LIN {X -0.159,Y -541.286,Z 1239.781,A 0.000,B 0.000,C 90.000,E1 176.674} C_DIS
LIN {X -0.066,Y -543.209,Z 1239.777,A 0.000,B 0.000,C 90.000,E1 175.812} C_DIS
LIN {X 0.150,Y -546.405,Z 1239.769,A 0.000,B 0.000,C 90.000,E1 174.375} C_DIS
LIN {X -0.133,Y -549.421,Z 1239.761,A 0.000,B 0.000,C 90.000,E1 172.996} C_DIS
LIN {X -0.115,Y -552.819,Z 1239.752,A 0.000,B 0.000,C 90.000,E1 171.310} C_DIS
LIN {X -0.232,Y -555.615,Z 1239.744,A 0.000,B 0.000,C 90.000,E1 169.926} C_DIS
LIN {X -0.113,Y -558.230,Z 1239.736,A 0.000,B 0.000,C 90.000,E1 168.522} C_DIS
LIN {X 0.206,Y -561.440,Z 1239.727,A 0.000,B 0.000,C 90.000,E1 166.825} C_DIS
LIN {X -0.219,Y -565.186,Z 1239.716,A 0.000,B 0.000,C 90.000,E1 164.936} C_DIS
LIN {X 0.264,Y -570.650,Z 1239.703,A 0.000,B 0.000,C 90.000,E1 162.417} C_DIS
LIN {X -0.154,Y -576.138,Z 1239.692,A 0.000,B 0.000,C 90.000,E1 160.550} C_DIS
LIN {X 0.101,Y -582.010,Z 1239.683,A 0.000,B 0.000,C 90.000,E1 158.901} C_DIS
LIN {X -0.130,Y -586.378,Z 1239.677,A 0.000,B 0.000,C 90.000,E1 157.847} C_DIS
LIN {X 0.033,Y -593.495,Z 1239.668,A 0.000,B 0.000,C 90.000,E1 156.230} C_DIS
LIN {X -0.128,Y -599.475,Z 1239.661,A 0.000,B 0.000,C 90.000,E1 154.921} C_DIS
LIN {X 0.061,Y -605.395,Z 1239.653,A 0.000,B 0.000,C 90.000,E1 153.589} C_DIS
LIN {X 0.125,Y -609.959,Z 1239.648,A 0.000,B 0.000,C 90.000,E1 152.538} C_DIS
LIN {X -0.028,Y -614.349,Z 1239.642,A 0.000,B 0.000,C 90.000,E1 151.513} C_DIS
LIN {X 0.169,Y -618.559,Z 1239.636,A 0.000,B 0.000,C 90.000,E1 150.461} C_DIS
LIN {X -0.124,Y -624.838,Z 1239.627,A 0.000,B 0.000,C 90.000,E1 148.948} C_DIS
LIN {X 0.004,Y -628.846,Z 1239.622,A 0.000,B 0.000,C 90.000,E1 147.916} C_DIS
LIN {X -0.147,Y -632.777,Z 1239.616,A 0.000,B 0.000,C 90.000,E1 146.914} C_DIS
LIN {X -0.050,Y -637.321,Z 1239.609,A 0.000,B 0.000,C 90.000,E1 145.642} C_DIS
LIN {X 0.260,Y -640.796,Z 1239.604,A 0.000,B 0.000,C 90.000,E1 144.609} C_DIS
LIN {X 0.090,Y -643.931,Z 1239.598,A 0.000,B 0.000,C 90.000,E1 143.623} C_DIS
LIN {X -0.137,Y -647.459,Z 1239.591,A 0.000,B 0.000,C 90.000,E1 142.396} C_DIS
LIN {X 0.168,Y -650.146,Z 1239.586,A 0.000,B 0.000,C 90.000,E1 141.376} C_DIS
LIN {X -0.411,Y -652.643,Z 1239.580,A 0.000,B 0.000,C 90.000,E1 140.436} C_DIS
LIN {X -0.144,Y -656.271,Z 1239.572,A 0.000,B 0.000,C 90.000,E1 138.933} C_DIS
LIN {X -0.300,Y -659.807,Z 1239.564,A 0.000,B 0.000,C 90.000,E1 137.472} C_DIS
LIN {X 0.078,Y -662.638,Z 1239.557,A 0.000,B 0.000,C 90.000,E1 136.215} C_DIS
LIN {X 0.026,Y -668.777,Z 1239.543,A 0.000,B 0.000,C 90.000,E1 133.785} C_DIS
LIN {X 0.118,Y -672.513,Z 1239.535,A 0.000,B 0.000,C 90.000,E1 132.324} C_DIS
LIN {X -0.219,Y -676.296,Z 1239.527,A 0.000,B 0.000,C 90.000,E1 130.906} C_DIS
LIN {X 0.096,Y -680.057,Z 1239.519,A 0.000,B 0.000,C 90.000,E1 129.439} C_DIS
LIN {X -0.040,Y -683.726,Z 1239.511,A 0.000,B 0.000,C 90.000,E1 128.016} C_DIS
LIN {X 0.382,Y -686.776,Z 1239.505,A 0.000,B 0.000,C 90.000,E1 126.790} C_DIS
LIN {X -0.148,Y -689.067,Z 1239.499,A 0.000,B 0.000,C 90.000,E1 125.884} C_DIS
LIN {X -0.009,Y -692.235,Z 1239.491,A 0.000,B 0.000,C 90.000,E1 124.452} C_DIS
LIN {X -0.020,Y -695.390,Z 1239.484,A 0.000,B 0.000,C 90.000,E1 123.038} C_DIS
LIN {X -0.103,Y -696.843,Z 1239.480,A 0.000,B 0.000,C 90.000,E1 122.339} C_DIS
LIN {X 0.324,Y -699.079,Z 1239.473,A 0.000,B 0.000,C 90.000,E1 121.131} C_DIS
LIN {X -0.174,Y -701.315,Z 1239.467,A 0.000,B 0.000,C 90.000,E1 120.001} C_DIS
LIN {X -0.028,Y -703.175,Z 1239.460,A 0.000,B 0.000,C 90.000,E1 118.821} C_DIS
LIN {X 0.198,Y -704.139,Z 1239.456,A 0.000,B 0.000,C 90.000,E1 118.103} C_DIS
LIN {X 0.093,Y -705.071,Z 1239.451,A 0.000,B 0.000,C 90.000,E1 117.180} C_DIS
LIN {X 0.011,Y -705.580,Z 1239.447,A 0.000,B 0.000,C 90.000,E1 116.488} C_DIS
LIN {X -0.058,Y -705.835,Z 1239.443,A 0.000,B 0.000,C 90.000,E1 115.796} C_DIS
LIN {X 0.180,Y -705.686,Z 1239.439,A 0.000,B 0.000,C 90.000,E1 115.079} C_DIS
LIN {X -0.178,Y -705.329,Z 1239.437,A 0.000,B 0.000,C 90.000,E1 114.643} C_DIS
LIN {X 0.108,Y -704.589,Z 1239.434,A 0.000,B 0.000,C 90.000,E1 114.155} C_DIS
LIN {X -0.249,Y -704.115,Z 1239.433,A 0.000,B 0.000,C 90.000,E1 113.951} C_DIS
LIN {X 0.174,Y -701.663,Z 1239.430,A 0.000,B 0.000,C 90.000,E1 113.334} C_DIS
LIN {X 0.312,Y -700.871,Z 1239.429,A 0.000,B 0.000,C 90.000,E1 113.206} C_DIS
LIN {X 0.025,Y -696.095,Z 1239.427,A 0.000,B 0.000,C 90.000,E1 112.770} C_DIS
LIN {X 0.195,Y -694.683,Z 1239.426,A 0.000,B 0.000,C 90.000,E1 112.642} C_DIS
LIN {X 0.362,Y -692.329,Z 1239.425,A 0.000,B 0.000,C 90.000,E1 112.514} C_DIS
LIN {X 0.074,Y -686.037,Z 1239.424,A 0.000,B 0.000,C 90.000,E1 112.333} C_DIS
LIN {X -0.305,Y -683.624,Z 1239.424,A 0.000,B 0.000,C 90.000,E1 112.333} C_DIS
LIN {X -0.206,Y -677.436,Z 1239.424,A 0.000,B 0.000,C 90.000,E1 112.280} C_DIS
LIN {X -0.236,Y -621.471,Z 1239.424,A 0.000,B 0.000,C 90.000,E1 112.280} C_DIS
LIN {X 0.222,Y -618.148,Z 1239.422,A 0.000,B 0.000,C 90.000,E1 112.025} C_DIS
LIN {X -0.340,Y -616.389,Z 1239.421,A 0.000,B 0.000,C 90.000,E1 111.844} C_DIS
LIN {X -0.383,Y -616.380,Z 1239.421,A 0.000,B 0.000,C 90.000,E1 111.844} C_DIS
LIN {X -0.170,Y -616.270,Z 1239.420,A 0.000,B 0.000,C 90.000,E1 111.663} C_DIS
LIN {X -0.183,Y -616.646,Z 1239.420,A 0.000,B 0.000,C 90.000,E1 111.535} C_DIS
LIN {X 0.334,Y -618.749,Z 1239.417,A 0.000,B 0.000,C 90.000,E1 110.972} C_DIS
LIN {X -0.173,Y -622.755,Z 1239.412,A 0.000,B 0.000,C 90.000,E1 110.248} C_DIS
LIN {X 0.173,Y -625.249,Z 1239.410,A 0.000,B 0.000,C 90.000,E1 109.704} C_DIS
LIN {X -0.063,Y -628.625,Z 1239.405,A 0.000,B 0.000,C 90.000,E1 108.960} C_DIS
LIN {X -0.179,Y -640.008,Z 1239.391,A 0.000,B 0.000,C 90.000,E1 106.441} C_DIS
LIN {X 0.284,Y -642.172,Z 1239.389,A 0.000,B 0.000,C 90.000,E1 105.898} C_DIS
LIN {X -0.032,Y -644.177,Z 1239.386,A 0.000,B 0.000,C 90.000,E1 105.426} C_DIS
LIN {X -0.334,Y -646.007,Z 1239.383,A 0.000,B 0.000,C 90.000,E1 104.954} C_DIS
LIN {X 0.004,Y -647.639,Z 1239.380,A 0.000,B 0.000,C 90.000,E1 104.426} C_DIS
LIN {X -0.116,Y -648.936,Z 1239.377,A 0.000,B 0.000,C 90.000,E1 103.939} C_DIS
LIN {X 0.110,Y -650.550,Z 1239.373,A 0.000,B 0.000,C 90.000,E1 103.175} C_DIS
LIN {X -0.152,Y -651.298,Z 1239.371,A 0.000,B 0.000,C 90.000,E1 102.703} C_DIS
LIN {X 0.354,Y -651.536,Z 1239.369,A 0.000,B 0.000,C 90.000,E1 102.411} C_DIS
LIN {X -0.039,Y -651.751,Z 1239.366,A 0.000,B 0.000,C 90.000,E1 101.951} C_DIS
LIN {X -0.293,Y -651.502,Z 1239.364,A 0.000,B 0.000,C 90.000,E1 101.478} C_DIS
LIN {X 0.088,Y -650.980,Z 1239.361,A 0.000,B 0.000,C 90.000,E1 100.950} C_DIS
LIN {X -0.044,Y -650.643,Z 1239.359,A 0.000,B 0.000,C 90.000,E1 100.715} C_DIS
LIN {X 0.210,Y -649.651,Z 1239.357,A 0.000,B 0.000,C 90.000,E1 100.197} C_DIS
LIN {X -0.065,Y -648.276,Z 1239.354,A 0.000,B 0.000,C 90.000,E1 99.726} C_DIS
LIN {X 0.180,Y -646.565,Z 1239.351,A 0.000,B 0.000,C 90.000,E1 99.208} C_DIS
LIN {X -0.219,Y -644.492,Z 1239.349,A 0.000,B 0.000,C 90.000,E1 98.746} C_DIS
LIN {X 0.136,Y -642.730,Z 1239.346,A 0.000,B 0.000,C 90.000,E1 98.341} C_DIS
LIN {X -0.156,Y -640.829,Z 1239.344,A 0.000,B 0.000,C 90.000,E1 97.992} C_DIS
LIN {X -0.137,Y -636.009,Z 1239.340,A 0.000,B 0.000,C 90.000,E1 97.239} C_DIS
LIN {X 0.167,Y -633.458,Z 1239.338,A 0.000,B 0.000,C 90.000,E1 96.834} C_DIS
LIN {X 0.173,Y -628.255,Z 1239.335,A 0.000,B 0.000,C 90.000,E1 96.201} C_DIS
LIN {X -0.191,Y -625.016,Z 1239.333,A 0.000,B 0.000,C 90.000,E1 95.853} C_DIS
LIN {X -0.164,Y -617.303,Z 1239.328,A 0.000,B 0.000,C 90.000,E1 95.106} C_DIS
LIN {X -0.222,Y -610.306,Z 1239.325,A 0.000,B 0.000,C 90.000,E1 94.531} C_DIS
LIN {X -0.057,Y -604.326,Z 1239.323,A 0.000,B 0.000,C 90.000,E1 94.073} C_DIS
LIN {X 0.042,Y -596.685,Z 1239.320,A 0.000,B 0.000,C 90.000,E1 93.555} C_DIS
LIN {X 0.187,Y -586.971,Z 1239.317,A 0.000,B 0.000,C 90.000,E1 92.980} C_DIS
LIN {X 0.126,Y -583.659,Z 1239.316,A 0.000,B 0.000,C 90.000,E1 92.808} C_DIS
LIN {X -0.203,Y -576.652,Z 1239.314,A 0.000,B 0.000,C 90.000,E1 92.522} C_DIS
LIN {X -0.045,Y -571.225,Z 1239.313,A 0.000,B 0.000,C 90.000,E1 92.293} C_DIS
LIN {X -0.061,Y -567.337,Z 1239.312,A 0.000,B 0.000,C 90.000,E1 92.064} C_DIS
LIN {X 0.145,Y -566.878,Z 1239.311,A 0.000,B 0.000,C 90.000,E1 92.007} C_DIS
LIN {X -0.002,Y -566.188,Z 1239.311,A 0.000,B 0.000,C 90.000,E1 91.892} C_DIS
LIN {X -0.093,Y -566.019,Z 1239.306,A 0.000,B 0.000,C 90.000,E1 91.146} C_DIS
LIN {X 0.157,Y -567.324,Z 1239.296,A 0.000,B 0.000,C 90.000,E1 89.198} C_DIS
LIN {X -0.118,Y -568.765,Z 1239.285,A 0.000,B 0.000,C 90.000,E1 87.306} C_DIS
LIN {X 0.130,Y -571.142,Z 1239.270,A 0.000,B 0.000,C 90.000,E1 84.546} C_DIS
LIN {X -0.097,Y -572.726,Z 1239.261,A 0.000,B 0.000,C 90.000,E1 82.932} C_DIS
LIN {X -0.221,Y -574.365,Z 1239.252,A 0.000,B 0.000,C 90.000,E1 81.310} C_DIS
LIN {X -0.065,Y -575.384,Z 1239.246,A 0.000,B 0.000,C 90.000,E1 80.208} C_DIS
LIN {X -0.258,Y -576.370,Z 1239.238,A 0.000,B 0.000,C 90.000,E1 78.870} C_DIS
LIN {X 0.106,Y -577.627,Z 1239.228,A 0.000,B 0.000,C 90.000,E1 76.937} C_DIS
LIN {X -0.148,Y -578.654,Z 1239.219,A 0.000,B 0.000,C 90.000,E1 75.338} C_DIS
LIN {X -0.008,Y -579.712,Z 1239.208,A 0.000,B 0.000,C 90.000,E1 73.433} C_DIS
LIN {X -0.105,Y -580.316,Z 1239.202,A 0.000,B 0.000,C 90.000,E1 72.362} C_DIS
LIN {X -0.131,Y -581.509,Z 1239.192,A 0.000,B 0.000,C 90.000,E1 70.477} C_DIS
LIN {X 0.012,Y -582.379,Z 1239.182,A 0.000,B 0.000,C 90.000,E1 68.847} C_DIS
LIN {X 0.321,Y -584.062,Z 1239.171,A 0.000,B 0.000,C 90.000,E1 66.666} C_DIS
LIN {X -0.262,Y -585.676,Z 1239.160,A 0.000,B 0.000,C 90.000,E1 64.845} C_DIS
LIN {X 0.114,Y -587.635,Z 1239.148,A 0.000,B 0.000,C 90.000,E1 62.666} C_DIS
LIN {X 0.237,Y -589.240,Z 1239.139,A 0.000,B 0.000,C 90.000,E1 61.051} C_DIS
LIN {X 0.161,Y -590.895,Z 1239.130,A 0.000,B 0.000,C 90.000,E1 59.459} C_DIS
LIN {X 0.227,Y -592.252,Z 1239.123,A 0.000,B 0.000,C 90.000,E1 58.122} C_DIS
LIN {X -0.080,Y -593.318,Z 1239.117,A 0.000,B 0.000,C 90.000,E1 57.089} C_DIS
LIN {X 0.228,Y -594.723,Z 1239.108,A 0.000,B 0.000,C 90.000,E1 55.468} C_DIS
LIN {X -0.087,Y -596.078,Z 1239.099,A 0.000,B 0.000,C 90.000,E1 53.909} C_DIS
LIN {X 0.229,Y -597.028,Z 1239.092,A 0.000,B 0.000,C 90.000,E1 52.557} C_DIS
LIN {X -0.149,Y -597.936,Z 1239.086,A 0.000,B 0.000,C 90.000,E1 51.537} C_DIS
LIN {X 0.088,Y -598.439,Z 1239.082,A 0.000,B 0.000,C 90.000,E1 50.723} C_DIS
LIN {X 0.124,Y -599.217,Z 1239.073,A 0.000,B 0.000,C 90.000,E1 49.138} C_DIS
LIN {X 0.156,Y -599.656,Z 1239.067,A 0.000,B 0.000,C 90.000,E1 48.081} C_DIS
LIN {X -0.041,Y -599.960,Z 1239.063,A 0.000,B 0.000,C 90.000,E1 47.310} C_DIS
LIN {X -0.239,Y -600.183,Z 1239.058,A 0.000,B 0.000,C 90.000,E1 46.539} C_DIS
LIN {X 0.199,Y -600.293,Z 1239.050,A 0.000,B 0.000,C 90.000,E1 44.919} C_DIS
LIN {X 0.210,Y -600.158,Z 1239.044,A 0.000,B 0.000,C 90.000,E1 43.866} C_DIS
LIN {X 0.033,Y -599.798,Z 1239.036,A 0.000,B 0.000,C 90.000,E1 42.567} C_DIS
LIN {X 0.024,Y -599.344,Z 1239.031,A 0.000,B 0.000,C 90.000,E1 41.515} C_DIS
LIN {X 0.286,Y -598.606,Z 1239.023,A 0.000,B 0.000,C 90.000,E1 40.172} C_DIS
LIN {X 0.070,Y -598.239,Z 1239.019,A 0.000,B 0.000,C 90.000,E1 39.402} C_DIS
LIN {X -0.066,Y -597.699,Z 1239.015,A 0.000,B 0.000,C 90.000,E1 38.624} C_DIS
LIN {X -0.070,Y -596.650,Z 1239.009,A 0.000,B 0.000,C 90.000,E1 37.569} C_DIS
LIN {X 0.013,Y -595.473,Z 1239.003,A 0.000,B 0.000,C 90.000,E1 36.503} C_DIS
LIN {X -0.140,Y -594.382,Z 1238.998,A 0.000,B 0.000,C 90.000,E1 35.724} C_DIS
LIN {X -0.089,Y -592.672,Z 1238.993,A 0.000,B 0.000,C 90.000,E1 34.659} C_DIS
LIN {X -0.118,Y -591.215,Z 1238.988,A 0.000,B 0.000,C 90.000,E1 33.865} C_DIS
LIN {X 0.295,Y -590.086,Z 1238.985,A 0.000,B 0.000,C 90.000,E1 33.293} C_DIS
LIN {X -0.053,Y -587.340,Z 1238.979,A 0.000,B 0.000,C 90.000,E1 32.260} C_DIS
LIN {X -0.121,Y -585.016,Z 1238.975,A 0.000,B 0.000,C 90.000,E1 31.465} C_DIS
LIN {X -0.207,Y -582.273,Z 1238.970,A 0.000,B 0.000,C 90.000,E1 30.669} C_DIS
LIN {X -0.182,Y -580.238,Z 1238.967,A 0.000,B 0.000,C 90.000,E1 30.129} C_DIS
LIN {X 0.185,Y -576.738,Z 1238.963,A 0.000,B 0.000,C 90.000,E1 29.283} C_DIS
LIN {X 0.242,Y -574.841,Z 1238.961,A 0.000,B 0.000,C 90.000,E1 28.871} C_DIS
LIN {X 0.372,Y -569.197,Z 1238.955,A 0.000,B 0.000,C 90.000,E1 27.769} C_DIS
LIN {X -0.066,Y -565.217,Z 1238.951,A 0.000,B 0.000,C 90.000,E1 27.129} C_DIS
LIN {X 0.124,Y -560.088,Z 1238.946,A 0.000,B 0.000,C 90.000,E1 26.283} C_DIS
LIN {X 0.114,Y -555.294,Z 1238.942,A 0.000,B 0.000,C 90.000,E1 25.591} C_DIS
LIN {X 0.179,Y -551.321,Z 1238.939,A 0.000,B 0.000,C 90.000,E1 25.027} C_DIS
LIN {X 0.097,Y -545.830,Z 1238.935,A 0.000,B 0.000,C 90.000,E1 24.335} C_DIS
LIN {X 0.223,Y -542.367,Z 1238.933,A 0.000,B 0.000,C 90.000,E1 23.898} C_DIS
LIN {X 0.140,Y -532.373,Z 1238.927,A 0.000,B 0.000,C 90.000,E1 22.770} C_DIS
LIN {X 0.215,Y -528.501,Z 1238.924,A 0.000,B 0.000,C 90.000,E1 22.333} C_DIS
LIN {X -0.131,Y -519.371,Z 1238.919,A 0.000,B 0.000,C 90.000,E1 21.408} C_DIS
LIN {X 0.117,Y -508.642,Z 1238.913,A 0.000,B 0.000,C 90.000,E1 20.301} C_DIS
LIN {X -0.303,Y -498.892,Z 1238.908,A 0.000,B 0.000,C 90.000,E1 19.396} C_DIS
LIN {X 0.252,Y -489.022,Z 1238.903,A 0.000,B 0.000,C 90.000,E1 18.417} C_DIS
LIN {X 0.134,Y -480.227,Z 1238.898,A 0.000,B 0.000,C 90.000,E1 17.638} C_DIS
LIN {X -0.082,Y -465.601,Z 1238.891,A 0.000,B 0.000,C 90.000,E1 16.370} C_DIS
LIN {X -0.175,Y -443.465,Z 1238.880,A 0.000,B 0.000,C 90.000,E1 14.356} C_DIS
LIN {X -0.151,Y -424.558,Z 1238.869,A 0.000,B 0.000,C 90.000,E1 12.479} C_DIS
LIN {X -0.208,Y -403.283,Z 1238.856,A 0.000,B 0.000,C 90.000,E1 10.141} C_DIS
LIN {X 0.008,Y -399.230,Z 1238.854,A 0.000,B 0.000,C 90.000,E1 9.613} C_DIS
LIN {X -0.165,Y -396.098,Z 1238.851,A 0.000,B 0.000,C 90.000,E1 9.208} C_DIS
LIN {X 0.169,Y -395.193,Z 1238.850,A 0.000,B 0.000,C 90.000,E1 8.973} C_DIS
LIN {X 0.133,Y -394.246,Z 1238.849,A 0.000,B 0.000,C 90.000,E1 8.746} C_DIS
LIN {X 0.095,Y -394.236,Z 1238.849,A 0.000,B 0.000,C 90.000,E1 8.746} C_DIS
LIN {X -0.015,Y -394.164,Z 1238.848,A 0.000,B 0.000,C 90.000,E1 8.624} C_DIS
LIN {X -0.053,Y -394.166,Z 1238.848,A 0.000,B 0.000,C 90.000,E1 8.624} C_DIS
LIN {X 0.054,Y -396.357,Z 1238.845,A 0.000,B 0.000,C 90.000,E1 8.106} C_DIS
LIN {X 0.009,Y -397.853,Z 1238.844,A 0.000,B 0.000,C 90.000,E1 7.936} C_DIS
LIN {X -0.119,Y -400.874,Z 1238.842,A 0.000,B 0.000,C 90.000,E1 7.644} C_DIS
LIN {X 0.079,Y -406.596,Z 1238.840,A 0.000,B 0.000,C 90.000,E1 7.182} C_DIS
LIN {X -0.195,Y -414.525,Z 1238.837,A 0.000,B 0.000,C 90.000,E1 6.663} C_DIS
LIN {X 0.109,Y -422.610,Z 1238.834,A 0.000,B 0.000,C 90.000,E1 6.030} C_DIS
LIN {X -0.031,Y -430.604,Z 1238.830,A 0.000,B 0.000,C 90.000,E1 5.454} C_DIS
LIN {X -0.034,Y -443.124,Z 1238.825,A 0.000,B 0.000,C 90.000,E1 4.473} C_DIS
LIN {X -0.210,Y -457.129,Z 1238.819,A 0.000,B 0.000,C 90.000,E1 3.383} C_DIS
LIN {X -0.016,Y -463.216,Z 1238.816,A 0.000,B 0.000,C 90.000,E1 2.865} C_DIS
LIN {X 0.078,Y -469.211,Z 1238.813,A 0.000,B 0.000,C 90.000,E1 2.350} C_DIS
LIN {X 0.196,Y -473.636,Z 1238.811,A 0.000,B 0.000,C 90.000,E1 1.949} C_DIS
LIN {X 0.117,Y -479.358,Z 1238.808,A 0.000,B 0.000,C 90.000,E1 1.432} C_DIS
LIN {X -0.201,Y -484.890,Z 1238.805,A 0.000,B 0.000,C 90.000,E1 0.917} C_DIS
LIN {X -0.067,Y -491.548,Z 1238.801,A 0.000,B 0.000,C 90.000,E1 0.172} C_DIS
LIN {X 0.082,Y -497.345,Z 1238.797,A 0.000,B 0.000,C 90.000,E1 359.484} C_DIS
LIN {X 0.034,Y -503.232,Z 1238.793,A 0.000,B 0.000,C 90.000,E1 358.740} C_DIS
LIN {X 0.052,Y -508.653,Z 1238.789,A 0.000,B 0.000,C 90.000,E1 357.993} C_DIS
LIN {X 0.076,Y -513.670,Z 1238.785,A 0.000,B 0.000,C 90.000,E1 357.249} C_DIS
LIN {X 0.167,Y -518.402,Z 1238.781,A 0.000,B 0.000,C 90.000,E1 356.502} C_DIS
LIN {X 0.076,Y -521.935,Z 1238.777,A 0.000,B 0.000,C 90.000,E1 355.927} C_DIS
LIN {X 0.208,Y -525.937,Z 1238.773,A 0.000,B 0.000,C 90.000,E1 355.184} C_DIS
LIN {X -0.062,Y -529.601,Z 1238.769,A 0.000,B 0.000,C 90.000,E1 354.489} C_DIS
LIN {X -0.071,Y -532.321,Z 1238.766,A 0.000,B 0.000,C 90.000,E1 353.913} C_DIS
LIN {X -0.060,Y -534.872,Z 1238.763,A 0.000,B 0.000,C 90.000,E1 353.337} C_DIS
LIN {X -0.034,Y -537.243,Z 1238.760,A 0.000,B 0.000,C 90.000,E1 352.761} C_DIS
LIN {X 0.068,Y -540.450,Z 1238.755,A 0.000,B 0.000,C 90.000,E1 351.894} C_DIS
LIN {X 0.202,Y -543.387,Z 1238.750,A 0.000,B 0.000,C 90.000,E1 351.027} C_DIS
LIN {X -0.080,Y -546.130,Z 1238.746,A 0.000,B 0.000,C 90.000,E1 350.208} C_DIS
LIN {X -0.223,Y -550.100,Z 1238.738,A 0.000,B 0.000,C 90.000,E1 348.814} C_DIS
LIN {X -0.197,Y -553.570,Z 1238.730,A 0.000,B 0.000,C 90.000,E1 347.409} C_DIS
LIN {X -0.112,Y -556.059,Z 1238.724,A 0.000,B 0.000,C 90.000,E1 346.284} C_DIS
LIN {X -0.128,Y -558.246,Z 1238.718,A 0.000,B 0.000,C 90.000,E1 345.172} C_DIS
LIN {X 0.173,Y -560.272,Z 1238.711,A 0.000,B 0.000,C 90.000,E1 344.031} C_DIS
LIN {X -0.184,Y -562.020,Z 1238.705,A 0.000,B 0.000,C 90.000,E1 342.960} C_DIS
LIN {X 0.180,Y -563.501,Z 1238.699,A 0.000,B 0.000,C 90.000,E1 341.819} C_DIS
LIN {X 0.028,Y -564.723,Z 1238.693,A 0.000,B 0.000,C 90.000,E1 340.732} C_DIS
LIN {X 0.084,Y -565.529,Z 1238.687,A 0.000,B 0.000,C 90.000,E1 339.625} C_DIS
LIN {X -0.177,Y -565.847,Z 1238.682,A 0.000,B 0.000,C 90.000,E1 338.827} C_DIS
LIN {X -0.244,Y -565.913,Z 1238.679,A 0.000,B 0.000,C 90.000,E1 338.284} C_DIS
LIN {X 0.232,Y -565.700,Z 1238.675,A 0.000,B 0.000,C 90.000,E1 337.411} C_DIS
LIN {X -0.036,Y -565.160,Z 1238.670,A 0.000,B 0.000,C 90.000,E1 336.613} C_DIS
LIN {X 0.238,Y -563.873,Z 1238.664,A 0.000,B 0.000,C 90.000,E1 335.485} C_DIS
LIN {X -0.143,Y -563.050,Z 1238.661,A 0.000,B 0.000,C 90.000,E1 334.973} C_DIS
LIN {X -0.214,Y -561.509,Z 1238.656,A 0.000,B 0.000,C 90.000,E1 334.152} C_DIS
LIN {X 0.244,Y -558.987,Z 1238.650,A 0.000,B 0.000,C 90.000,E1 332.999} C_DIS
LIN {X 0.041,Y -558.330,Z 1238.649,A 0.000,B 0.000,C 90.000,E1 332.743} C_DIS
LIN {X -0.046,Y -554.735,Z 1238.642,A 0.000,B 0.000,C 90.000,E1 331.641} C_DIS
LIN {X 0.043,Y -551.366,Z 1238.638,A 0.000,B 0.000,C 90.000,E1 330.795} C_DIS
LIN {X -0.148,Y -548.734,Z 1238.635,A 0.000,B 0.000,C 90.000,E1 330.255} C_DIS
LIN {X 0.116,Y -545.883,Z 1238.632,A 0.000,B 0.000,C 90.000,E1 329.665} C_DIS
LIN {X -0.111,Y -542.741,Z 1238.628,A 0.000,B 0.000,C 90.000,E1 329.125} C_DIS
LIN {X 0.113,Y -537.269,Z 1238.624,A 0.000,B 0.000,C 90.000,E1 328.250} C_DIS
LIN {X 0.134,Y -532.378,Z 1238.620,A 0.000,B 0.000,C 90.000,E1 327.533} C_DIS
LIN {X -0.209,Y -526.129,Z 1238.615,A 0.000,B 0.000,C 90.000,E1 326.707} C_DIS
LIN {X -0.060,Y -518.520,Z 1238.609,A 0.000,B 0.000,C 90.000,E1 325.674} C_DIS
LIN {X 0.147,Y -514.711,Z 1238.606,A 0.000,B 0.000,C 90.000,E1 325.102} C_DIS
LIN {X -0.051,Y -511.652,Z 1238.603,A 0.000,B 0.000,C 90.000,E1 324.609} C_DIS
LIN {X -0.240,Y -508.815,Z 1238.600,A 0.000,B 0.000,C 90.000,E1 323.989} C_DIS
LIN {X 0.113,Y -506.962,Z 1238.596,A 0.000,B 0.000,C 90.000,E1 323.210} C_DIS
LIN {X -0.082,Y -506.057,Z 1238.592,A 0.000,B 0.000,C 90.000,E1 322.637} C_DIS
LIN {X 0.024,Y -505.470,Z 1238.589,A 0.000,B 0.000,C 90.000,E1 322.029} C_DIS
LIN {X -0.182,Y -505.207,Z 1238.586,A 0.000,B 0.000,C 90.000,E1 321.457} C_DIS
LIN {X -0.173,Y -506.208,Z 1238.571,A 0.000,B 0.000,C 90.000,E1 318.771} C_DIS
LIN {X 0.292,Y -506.801,Z 1238.563,A 0.000,B 0.000,C 90.000,E1 317.229} C_DIS
LIN {X -0.324,Y -507.316,Z 1238.554,A 0.000,B 0.000,C 90.000,E1 315.810} C_DIS
LIN {X -0.105,Y -507.935,Z 1238.543,A 0.000,B 0.000,C 90.000,E1 313.704} C_DIS
LIN {X 0.144,Y -508.691,Z 1238.531,A 0.000,B 0.000,C 90.000,E1 311.595} C_DIS
LIN {X 0.317,Y -509.214,Z 1238.523,A 0.000,B 0.000,C 90.000,E1 310.092} C_DIS
LIN {X 0.178,Y -509.639,Z 1238.515,A 0.000,B 0.000,C 90.000,E1 308.624} C_DIS
LIN {X 0.046,Y -510.089,Z 1238.506,A 0.000,B 0.000,C 90.000,E1 307.156} C_DIS
LIN {X 0.109,Y -510.410,Z 1238.500,A 0.000,B 0.000,C 90.000,E1 305.964} C_DIS
LIN {X 0.094,Y -510.717,Z 1238.492,A 0.000,B 0.000,C 90.000,E1 304.485} C_DIS
LIN {X 0.073,Y -511.002,Z 1238.484,A 0.000,B 0.000,C 90.000,E1 303.007} C_DIS
LIN {X -0.072,Y -511.155,Z 1238.475,A 0.000,B 0.000,C 90.000,E1 301.544} C_DIS
LIN {X 0.137,Y -511.238,Z 1238.465,A 0.000,B 0.000,C 90.000,E1 299.745} C_DIS
LIN {X -0.003,Y -511.239,Z 1238.457,A 0.000,B 0.000,C 90.000,E1 298.281} C_DIS
LIN {X 0.054,Y -511.208,Z 1238.449,A 0.000,B 0.000,C 90.000,E1 296.796} C_DIS
LIN {X 0.068,Y -511.329,Z 1238.434,A 0.000,B 0.000,C 90.000,E1 294.131} C_DIS
LIN {X 0.046,Y -511.394,Z 1238.428,A 0.000,B 0.000,C 90.000,E1 292.950} C_DIS
LIN {X 0.136,Y -510.947,Z 1238.419,A 0.000,B 0.000,C 90.000,E1 291.461} C_DIS
LIN {X -0.079,Y -510.463,Z 1238.413,A 0.000,B 0.000,C 90.000,E1 290.301} C_DIS
LIN {X -0.212,Y -509.464,Z 1238.400,A 0.000,B 0.000,C 90.000,E1 287.946} C_DIS
LIN {X -0.067,Y -509.112,Z 1238.395,A 0.000,B 0.000,C 90.000,E1 287.040} C_DIS
LIN {X 0.003,Y -508.188,Z 1238.383,A 0.000,B 0.000,C 90.000,E1 284.954} C_DIS
LIN {X 0.010,Y -507.302,Z 1238.375,A 0.000,B 0.000,C 90.000,E1 283.467} C_DIS
LIN {X -0.138,Y -506.650,Z 1238.370,A 0.000,B 0.000,C 90.000,E1 282.591} C_DIS
LIN {X 0.209,Y -506.076,Z 1238.365,A 0.000,B 0.000,C 90.000,E1 281.658} C_DIS
LIN {X 0.216,Y -504.023,Z 1238.350,A 0.000,B 0.000,C 90.000,E1 278.973} C_DIS
LIN {X -0.244,Y -503.117,Z 1238.342,A 0.000,B 0.000,C 90.000,E1 277.530} C_DIS
LIN {X 0.005,Y -501.816,Z 1238.328,A 0.000,B 0.000,C 90.000,E1 275.106} C_DIS
LIN {X -0.164,Y -500.807,Z 1238.318,A 0.000,B 0.000,C 90.000,E1 273.326} C_DIS
LIN {X -0.131,Y -500.000,Z 1238.312,A 0.000,B 0.000,C 90.000,E1 272.121} C_DIS
LIN {X -0.115,Y -499.040,Z 1238.305,A 0.000,B 0.000,C 90.000,E1 270.917} C_DIS
LIN {X -0.016,Y -497.609,Z 1238.293,A 0.000,B 0.000,C 90.000,E1 268.797} C_DIS
LIN {X 0.099,Y -497.010,Z 1238.288,A 0.000,B 0.000,C 90.000,E1 267.879} C_DIS
LIN {X -0.062,Y -496.196,Z 1238.280,A 0.000,B 0.000,C 90.000,E1 266.388} C_DIS
LIN {X 0.130,Y -495.162,Z 1238.270,A 0.000,B 0.000,C 90.000,E1 264.552} C_DIS
LIN {X -0.099,Y -493.875,Z 1238.260,A 0.000,B 0.000,C 90.000,E1 262.761} C_DIS
LIN {X -0.079,Y -492.806,Z 1238.253,A 0.000,B 0.000,C 90.000,E1 261.546} C_DIS
LIN {X -0.120,Y -490.157,Z 1238.238,A 0.000,B 0.000,C 90.000,E1 258.814} C_DIS
LIN {X 0.167,Y -488.574,Z 1238.226,A 0.000,B 0.000,C 90.000,E1 256.645} C_DIS
LIN {X 0.045,Y -487.272,Z 1238.214,A 0.000,B 0.000,C 90.000,E1 254.519} C_DIS
LIN {X 0.150,Y -485.968,Z 1238.202,A 0.000,B 0.000,C 90.000,E1 252.362} C_DIS
LIN {X -0.085,Y -484.912,Z 1238.190,A 0.000,B 0.000,C 90.000,E1 250.242} C_DIS
LIN {X -0.212,Y -484.287,Z 1238.183,A 0.000,B 0.000,C 90.000,E1 249.028} C_DIS
LIN {X -0.171,Y -483.475,Z 1238.175,A 0.000,B 0.000,C 90.000,E1 247.486} C_DIS
LIN {X 0.040,Y -482.481,Z 1238.166,A 0.000,B 0.000,C 90.000,E1 245.921} C_DIS
LIN {X -0.003,Y -481.068,Z 1238.156,A 0.000,B 0.000,C 90.000,E1 244.076} C_DIS
LIN {X -0.063,Y -479.930,Z 1238.147,A 0.000,B 0.000,C 90.000,E1 242.538} C_DIS
LIN {X 0.078,Y -478.591,Z 1238.139,A 0.000,B 0.000,C 90.000,E1 240.973} C_DIS
LIN {X -0.011,Y -477.472,Z 1238.132,A 0.000,B 0.000,C 90.000,E1 239.744} C_DIS
LIN {X 0.087,Y -475.588,Z 1238.122,A 0.000,B 0.000,C 90.000,E1 237.867} C_DIS
LIN {X 0.000,Y -473.771,Z 1238.111,A 0.000,B 0.000,C 90.000,E1 236.008} C_DIS
LIN {X 0.144,Y -472.113,Z 1238.101,A 0.000,B 0.000,C 90.000,E1 234.116} C_DIS
LIN {X -0.136,Y -470.493,Z 1238.090,A 0.000,B 0.000,C 90.000,E1 232.271} C_DIS
LIN {X -0.112,Y -468.614,Z 1238.078,A 0.000,B 0.000,C 90.000,E1 230.070} C_DIS
LIN {X 0.112,Y -466.861,Z 1238.066,A 0.000,B 0.000,C 90.000,E1 227.838} C_DIS
LIN {X -0.116,Y -465.418,Z 1238.055,A 0.000,B 0.000,C 90.000,E1 225.972} C_DIS
LIN {X -0.013,Y -463.787,Z 1238.034,A 0.000,B 0.000,C 90.000,E1 222.162} C_DIS
LIN {X -0.093,Y -465.130,Z 1237.997,A 0.000,B 0.000,C 90.000,E1 215.518} C_DIS
LIN {X 0.033,Y -468.440,Z 1237.973,A 0.000,B 0.000,C 90.000,E1 211.082} C_DIS
LIN {X -0.088,Y -472.228,Z 1237.954,A 0.000,B 0.000,C 90.000,E1 207.641} C_DIS
LIN {X -0.139,Y -474.591,Z 1237.943,A 0.000,B 0.000,C 90.000,E1 205.771} C_DIS
LIN {X -0.009,Y -479.495,Z 1237.924,A 0.000,B 0.000,C 90.000,E1 202.333} C_DIS
LIN {X -0.197,Y -485.542,Z 1237.905,A 0.000,B 0.000,C 90.000,E1 198.960} C_DIS
LIN {X -0.173,Y -492.217,Z 1237.888,A 0.000,B 0.000,C 90.000,E1 195.898} C_DIS
LIN {X -0.060,Y -496.543,Z 1237.878,A 0.000,B 0.000,C 90.000,E1 194.064} C_DIS
LIN {X 0.116,Y -500.278,Z 1237.870,A 0.000,B 0.000,C 90.000,E1 192.535} C_DIS
LIN {X 0.145,Y -505.606,Z 1237.858,A 0.000,B 0.000,C 90.000,E1 190.433} C_DIS
LIN {X -0.276,Y -511.238,Z 1237.847,A 0.000,B 0.000,C 90.000,E1 188.398} C_DIS
LIN {X -0.014,Y -515.254,Z 1237.838,A 0.000,B 0.000,C 90.000,E1 186.891} C_DIS
LIN {X 0.121,Y -520.743,Z 1237.827,A 0.000,B 0.000,C 90.000,E1 184.821} C_DIS
LIN {X -0.070,Y -524.642,Z 1237.819,A 0.000,B 0.000,C 90.000,E1 183.383} C_DIS
LIN {X -0.222,Y -528.511,Z 1237.811,A 0.000,B 0.000,C 90.000,E1 181.949} C_DIS
LIN {X 0.253,Y -530.814,Z 1237.806,A 0.000,B 0.000,C 90.000,E1 181.031} C_DIS
LIN {X 0.198,Y -534.608,Z 1237.798,A 0.000,B 0.000,C 90.000,E1 179.599} C_DIS
LIN {X 0.201,Y -537.567,Z 1237.792,A 0.000,B 0.000,C 90.000,E1 178.453} C_DIS
LIN {X 0.260,Y -540.380,Z 1237.785,A 0.000,B 0.000,C 90.000,E1 177.306} C_DIS
LIN {X -0.180,Y -543.140,Z 1237.779,A 0.000,B 0.000,C 90.000,E1 176.216} C_DIS
LIN {X 0.138,Y -547.659,Z 1237.768,A 0.000,B 0.000,C 90.000,E1 174.204} C_DIS
LIN {X -0.060,Y -550.679,Z 1237.760,A 0.000,B 0.000,C 90.000,E1 172.818} C_DIS
LIN {X -0.087,Y -554.231,Z 1237.751,A 0.000,B 0.000,C 90.000,E1 171.141} C_DIS
LIN {X -0.089,Y -557.072,Z 1237.743,A 0.000,B 0.000,C 90.000,E1 169.746} C_DIS
LIN {X 0.065,Y -559.775,Z 1237.735,A 0.000,B 0.000,C 90.000,E1 168.342} C_DIS
LIN {X -0.124,Y -563.074,Z 1237.726,A 0.000,B 0.000,C 90.000,E1 166.700} C_DIS
LIN {X -0.118,Y -566.420,Z 1237.717,A 0.000,B 0.000,C 90.000,E1 165.046} C_DIS
LIN {X 0.249,Y -572.000,Z 1237.703,A 0.000,B 0.000,C 90.000,E1 162.543} C_DIS
LIN {X -0.143,Y -577.479,Z 1237.693,A 0.000,B 0.000,C 90.000,E1 160.678} C_DIS
LIN {X 0.137,Y -583.215,Z 1237.684,A 0.000,B 0.000,C 90.000,E1 159.028} C_DIS
LIN {X 0.221,Y -589.838,Z 1237.675,A 0.000,B 0.000,C 90.000,E1 157.411} C_DIS
LIN {X 0.005,Y -595.701,Z 1237.667,A 0.000,B 0.000,C 90.000,E1 156.102} C_DIS
LIN {X -0.121,Y -601.578,Z 1237.660,A 0.000,B 0.000,C 90.000,E1 154.793} C_DIS
LIN {X 0.156,Y -606.242,Z 1237.654,A 0.000,B 0.000,C 90.000,E1 153.717} C_DIS
LIN {X -0.049,Y -610.732,Z 1237.648,A 0.000,B 0.000,C 90.000,E1 152.692} C_DIS
LIN {X 0.091,Y -615.025,Z 1237.643,A 0.000,B 0.000,C 90.000,E1 151.641} C_DIS
LIN {X 0.299,Y -619.154,Z 1237.637,A 0.000,B 0.000,C 90.000,E1 150.589} C_DIS
LIN {X 0.021,Y -625.228,Z 1237.628,A 0.000,B 0.000,C 90.000,E1 149.076} C_DIS
LIN {X 0.166,Y -630.145,Z 1237.621,A 0.000,B 0.000,C 90.000,E1 147.788} C_DIS
LIN {X 0.031,Y -633.889,Z 1237.616,A 0.000,B 0.000,C 90.000,E1 146.786} C_DIS
LIN {X 0.263,Y -636.554,Z 1237.611,A 0.000,B 0.000,C 90.000,E1 146.008} C_DIS
LIN {X 0.037,Y -640.008,Z 1237.606,A 0.000,B 0.000,C 90.000,E1 145.022} C_DIS
LIN {X -0.058,Y -641.677,Z 1237.603,A 0.000,B 0.000,C 90.000,E1 144.529} C_DIS
LIN {X -0.218,Y -644.675,Z 1237.597,A 0.000,B 0.000,C 90.000,E1 143.543} C_DIS
LIN {X 0.082,Y -648.118,Z 1237.590,A 0.000,B 0.000,C 90.000,E1 142.271} C_DIS
LIN {X -0.086,Y -651.340,Z 1237.584,A 0.000,B 0.000,C 90.000,E1 141.045} C_DIS
LIN {X -0.297,Y -654.312,Z 1237.577,A 0.000,B 0.000,C 90.000,E1 139.828} C_DIS
LIN {X -0.411,Y -656.689,Z 1237.571,A 0.000,B 0.000,C 90.000,E1 138.852} C_DIS
LIN {X -0.087,Y -659.620,Z 1237.564,A 0.000,B 0.000,C 90.000,E1 137.595} C_DIS
LIN {X -0.175,Y -663.007,Z 1237.556,A 0.000,B 0.000,C 90.000,E1 136.134} C_DIS
LIN {X -0.218,Y -669.111,Z 1237.543,A 0.000,B 0.000,C 90.000,E1 133.704} C_DIS
LIN {X -0.120,Y -672.855,Z 1237.535,A 0.000,B 0.000,C 90.000,E1 132.243} C_DIS
LIN {X 0.058,Y -676.610,Z 1237.527,A 0.000,B 0.000,C 90.000,E1 130.782} C_DIS
LIN {X -0.136,Y -680.348,Z 1237.519,A 0.000,B 0.000,C 90.000,E1 129.358} C_DIS
LIN {X -0.117,Y -684.611,Z 1237.509,A 0.000,B 0.000,C 90.000,E1 127.684} C_DIS
LIN {X -0.226,Y -687.628,Z 1237.503,A 0.000,B 0.000,C 90.000,E1 126.503} C_DIS
LIN {X -0.378,Y -689.328,Z 1237.499,A 0.000,B 0.000,C 90.000,E1 125.804} C_DIS
LIN {X 0.332,Y -692.498,Z 1237.491,A 0.000,B 0.000,C 90.000,E1 124.326} C_DIS
LIN {X 0.099,Y -695.153,Z 1237.484,A 0.000,B 0.000,C 90.000,E1 123.166} C_DIS
LIN {X 0.255,Y -697.081,Z 1237.479,A 0.000,B 0.000,C 90.000,E1 122.212} C_DIS
LIN {X 0.348,Y -699.778,Z 1237.471,A 0.000,B 0.000,C 90.000,E1 120.797} C_DIS
LIN {X 0.199,Y -701.523,Z 1237.466,A 0.000,B 0.000,C 90.000,E1 119.873} C_DIS
LIN {X -0.265,Y -703.436,Z 1237.460,A 0.000,B 0.000,C 90.000,E1 118.743} C_DIS
LIN {X 0.244,Y -704.592,Z 1237.454,A 0.000,B 0.000,C 90.000,E1 117.769} C_DIS
LIN {X -0.181,Y -705.446,Z 1237.449,A 0.000,B 0.000,C 90.000,E1 116.873} C_DIS
LIN {X 0.058,Y -705.814,Z 1237.445,A 0.000,B 0.000,C 90.000,E1 116.155} C_DIS
LIN {X -0.304,Y -705.935,Z 1237.443,A 0.000,B 0.000,C 90.000,E1 115.720} C_DIS
LIN {X -0.369,Y -705.725,Z 1237.439,A 0.000,B 0.000,C 90.000,E1 115.027} C_DIS
LIN {X 0.211,Y -705.341,Z 1237.436,A 0.000,B 0.000,C 90.000,E1 114.515} C_DIS
LIN {X -0.146,Y -704.549,Z 1237.434,A 0.000,B 0.000,C 90.000,E1 114.079} C_DIS
LIN {X 0.139,Y -703.840,Z 1237.432,A 0.000,B 0.000,C 90.000,E1 113.823} C_DIS
LIN {X -0.225,Y -701.803,Z 1237.430,A 0.000,B 0.000,C 90.000,E1 113.387} C_DIS
LIN {X -0.087,Y -701.068,Z 1237.429,A 0.000,B 0.000,C 90.000,E1 113.259} C_DIS
LIN {X -0.089,Y -698.721,Z 1237.428,A 0.000,B 0.000,C 90.000,E1 113.025} C_DIS
LIN {X -0.180,Y -695.031,Z 1237.426,A 0.000,B 0.000,C 90.000,E1 112.695} C_DIS
LIN {X -0.228,Y -693.057,Z 1237.425,A 0.000,B 0.000,C 90.000,E1 112.589} C_DIS
LIN {X 0.126,Y -686.215,Z 1237.424,A 0.000,B 0.000,C 90.000,E1 112.333} C_DIS
LIN {X -0.126,Y -685.182,Z 1237.424,A 0.000,B 0.000,C 90.000,E1 112.333} C_DIS
LIN {X -0.199,Y -677.161,Z 1237.424,A 0.000,B 0.000,C 90.000,E1 112.280} C_DIS
LIN {X -0.229,Y -620.472,Z 1237.424,A 0.000,B 0.000,C 90.000,E1 112.280} C_DIS
LIN {X 0.192,Y -617.806,Z 1237.423,A 0.000,B 0.000,C 90.000,E1 112.078} C_DIS
LIN {X -0.236,Y -616.859,Z 1237.422,A 0.000,B 0.000,C 90.000,E1 112.025} C_DIS
LIN {X -0.368,Y -615.087,Z 1237.421,A 0.000,B 0.000,C 90.000,E1 111.844} C_DIS
LIN {X 0.311,Y -614.938,Z 1237.421,A 0.000,B 0.000,C 90.000,E1 111.716} C_DIS
LIN {X -0.202,Y -614.914,Z 1237.420,A 0.000,B 0.000,C 90.000,E1 111.663} C_DIS
LIN {X -0.059,Y -615.601,Z 1237.419,A 0.000,B 0.000,C 90.000,E1 111.408} C_DIS
LIN {X -0.349,Y -617.782,Z 1237.416,A 0.000,B 0.000,C 90.000,E1 110.918} C_DIS
LIN {X -0.324,Y -620.311,Z 1237.413,A 0.000,B 0.000,C 90.000,E1 110.429} C_DIS
LIN {X -0.008,Y -623.432,Z 1237.410,A 0.000,B 0.000,C 90.000,E1 109.758} C_DIS
LIN {X 0.327,Y -626.747,Z 1237.406,A 0.000,B 0.000,C 90.000,E1 108.960} C_DIS
LIN {X 0.289,Y -631.542,Z 1237.399,A 0.000,B 0.000,C 90.000,E1 107.819} C_DIS
LIN {X -0.075,Y -635.615,Z 1237.394,A 0.000,B 0.000,C 90.000,E1 106.968} C_DIS
LIN {X -0.167,Y -640.139,Z 1237.389,A 0.000,B 0.000,C 90.000,E1 105.969} C_DIS
LIN {X -0.159,Y -641.185,Z 1237.387,A 0.000,B 0.000,C 90.000,E1 105.717} C_DIS
LIN {X -0.017,Y -643.975,Z 1237.383,A 0.000,B 0.000,C 90.000,E1 104.954} C_DIS
LIN {X -0.319,Y -645.507,Z 1237.380,A 0.000,B 0.000,C 90.000,E1 104.481} C_DIS
LIN {X 0.017,Y -646.945,Z 1237.378,A 0.000,B 0.000,C 90.000,E1 103.953} C_DIS
LIN {X 0.030,Y -647.523,Z 1237.376,A 0.000,B 0.000,C 90.000,E1 103.703} C_DIS
LIN {X 0.379,Y -648.467,Z 1237.373,A 0.000,B 0.000,C 90.000,E1 103.175} C_DIS
LIN {X -0.173,Y -649.559,Z 1237.369,A 0.000,B 0.000,C 90.000,E1 102.479} C_DIS
LIN {X 0.197,Y -649.786,Z 1237.367,A 0.000,B 0.000,C 90.000,E1 101.951} C_DIS
LIN {X -0.069,Y -649.528,Z 1237.364,A 0.000,B 0.000,C 90.000,E1 101.478} C_DIS
LIN {X 0.159,Y -648.612,Z 1237.360,A 0.000,B 0.000,C 90.000,E1 100.715} C_DIS
LIN {X -0.239,Y -647.597,Z 1237.357,A 0.000,B 0.000,C 90.000,E1 100.254} C_DIS
LIN {X 0.111,Y -646.208,Z 1237.354,A 0.000,B 0.000,C 90.000,E1 99.726} C_DIS
LIN {X -0.295,Y -644.508,Z 1237.351,A 0.000,B 0.000,C 90.000,E1 99.265} C_DIS
LIN {X -0.070,Y -642.452,Z 1237.349,A 0.000,B 0.000,C 90.000,E1 98.746} C_DIS
LIN {X -0.232,Y -641.312,Z 1237.347,A 0.000,B 0.000,C 90.000,E1 98.511} C_DIS
LIN {X -0.074,Y -637.841,Z 1237.344,A 0.000,B 0.000,C 90.000,E1 97.871} C_DIS
LIN {X -0.032,Y -633.863,Z 1237.340,A 0.000,B 0.000,C 90.000,E1 97.239} C_DIS
LIN {X 0.259,Y -631.201,Z 1237.338,A 0.000,B 0.000,C 90.000,E1 96.834} C_DIS
LIN {X 0.246,Y -625.976,Z 1237.335,A 0.000,B 0.000,C 90.000,E1 96.201} C_DIS
LIN {X -0.116,Y -622.416,Z 1237.333,A 0.000,B 0.000,C 90.000,E1 95.853} C_DIS
LIN {X 0.076,Y -617.407,Z 1237.330,A 0.000,B 0.000,C 90.000,E1 95.334} C_DIS
LIN {X -0.067,Y -610.497,Z 1237.326,A 0.000,B 0.000,C 90.000,E1 94.759} C_DIS
LIN {X 0.129,Y -603.034,Z 1237.323,A 0.000,B 0.000,C 90.000,E1 94.188} C_DIS
LIN {X -0.281,Y -595.216,Z 1237.321,A 0.000,B 0.000,C 90.000,E1 93.726} C_DIS
LIN {X 0.287,Y -584.228,Z 1237.317,A 0.000,B 0.000,C 90.000,E1 93.037} C_DIS
LIN {X 0.296,Y -580.414,Z 1237.316,A 0.000,B 0.000,C 90.000,E1 92.865} C_DIS
LIN {X -0.026,Y -571.859,Z 1237.314,A 0.000,B 0.000,C 90.000,E1 92.522} C_DIS
LIN {X 0.085,Y -566.784,Z 1237.313,A 0.000,B 0.000,C 90.000,E1 92.236} C_DIS
LIN {X 0.042,Y -566.759,Z 1237.313,A 0.000,B 0.000,C 90.000,E1 92.236} C_DIS
LIN {X -0.157,Y -566.349,Z 1237.312,A 0.000,B 0.000,C 90.000,E1 92.178} C_DIS
LIN {X 0.073,Y -565.918,Z 1237.311,A 0.000,B 0.000,C 90.000,E1 91.949} C_DIS
LIN {X 0.204,Y -565.846,Z 1237.309,A 0.000,B 0.000,C 90.000,E1 91.661} C_DIS
LIN {X -0.021,Y -566.103,Z 1237.305,A 0.000,B 0.000,C 90.000,E1 90.859} C_DIS
LIN {X 0.113,Y -567.281,Z 1237.296,A 0.000,B 0.000,C 90.000,E1 89.198} C_DIS
LIN {X -0.163,Y -568.704,Z 1237.285,A 0.000,B 0.000,C 90.000,E1 87.306} C_DIS
LIN {X -0.211,Y -570.516,Z 1237.273,A 0.000,B 0.000,C 90.000,E1 85.122} C_DIS
LIN {X 0.117,Y -572.128,Z 1237.264,A 0.000,B 0.000,C 90.000,E1 83.451} C_DIS
LIN {X 0.098,Y -574.013,Z 1237.253,A 0.000,B 0.000,C 90.000,E1 81.546} C_DIS
LIN {X -0.118,Y -575.259,Z 1237.246,A 0.000,B 0.000,C 90.000,E1 80.208} C_DIS
LIN {X 0.253,Y -576.231,Z 1237.238,A 0.000,B 0.000,C 90.000,E1 78.814} C_DIS
LIN {X 0.048,Y -577.492,Z 1237.228,A 0.000,B 0.000,C 90.000,E1 76.937} C_DIS
LIN {X -0.209,Y -578.504,Z 1237.219,A 0.000,B 0.000,C 90.000,E1 75.338} C_DIS
LIN {X 0.109,Y -579.394,Z 1237.209,A 0.000,B 0.000,C 90.000,E1 73.685} C_DIS
LIN {X 0.173,Y -580.032,Z 1237.203,A 0.000,B 0.000,C 90.000,E1 72.598} C_DIS
LIN {X 0.345,Y -581.356,Z 1237.192,A 0.000,B 0.000,C 90.000,E1 70.423} C_DIS
LIN {X -0.032,Y -583.453,Z 1237.174,A 0.000,B 0.000,C 90.000,E1 67.230} C_DIS
LIN {X -0.098,Y -585.074,Z 1237.163,A 0.000,B 0.000,C 90.000,E1 65.357} C_DIS
LIN {X -0.296,Y -586.436,Z 1237.154,A 0.000,B 0.000,C 90.000,E1 63.768} C_DIS
LIN {X 0.027,Y -587.511,Z 1237.148,A 0.000,B 0.000,C 90.000,E1 62.666} C_DIS
LIN {X 0.147,Y -589.118,Z 1237.139,A 0.000,B 0.000,C 90.000,E1 61.051} C_DIS
LIN {X 0.070,Y -590.781,Z 1237.130,A 0.000,B 0.000,C 90.000,E1 59.459} C_DIS
LIN {X 0.132,Y -592.121,Z 1237.123,A 0.000,B 0.000,C 90.000,E1 58.122} C_DIS
LIN {X -0.289,Y -593.388,Z 1237.116,A 0.000,B 0.000,C 90.000,E1 56.834} C_DIS
LIN {X 0.129,Y -594.574,Z 1237.108,A 0.000,B 0.000,C 90.000,E1 55.468} C_DIS
LIN {X 0.067,Y -595.681,Z 1237.101,A 0.000,B 0.000,C 90.000,E1 54.149} C_DIS
LIN {X -0.338,Y -596.505,Z 1237.095,A 0.000,B 0.000,C 90.000,E1 53.130} C_DIS
LIN {X -0.258,Y -597.767,Z 1237.086,A 0.000,B 0.000,C 90.000,E1 51.537} C_DIS
LIN {X -0.022,Y -598.279,Z 1237.082,A 0.000,B 0.000,C 90.000,E1 50.723} C_DIS
LIN {X 0.010,Y -599.028,Z 1237.073,A 0.000,B 0.000,C 90.000,E1 49.138} C_DIS
LIN {X 0.040,Y -599.500,Z 1237.067,A 0.000,B 0.000,C 90.000,E1 48.081} C_DIS
LIN {X -0.160,Y -599.789,Z 1237.063,A 0.000,B 0.000,C 90.000,E1 47.310} C_DIS
LIN {X 0.053,Y -600.011,Z 1237.058,A 0.000,B 0.000,C 90.000,E1 46.500} C_DIS
LIN {X 0.075,Y -600.119,Z 1237.050,A 0.000,B 0.000,C 90.000,E1 44.919} C_DIS
LIN {X 0.084,Y -599.972,Z 1237.044,A 0.000,B 0.000,C 90.000,E1 43.866} C_DIS
LIN {X 0.309,Y -599.605,Z 1237.036,A 0.000,B 0.000,C 90.000,E1 42.528} C_DIS
LIN {X -0.108,Y -599.125,Z 1237.031,A 0.000,B 0.000,C 90.000,E1 41.515} C_DIS
LIN {X 0.151,Y -598.396,Z 1237.023,A 0.000,B 0.000,C 90.000,E1 40.172} C_DIS
LIN {X -0.067,Y -598.023,Z 1237.019,A 0.000,B 0.000,C 90.000,E1 39.402} C_DIS
LIN {X -0.205,Y -597.473,Z 1237.015,A 0.000,B 0.000,C 90.000,E1 38.624} C_DIS
LIN {X 0.261,Y -596.412,Z 1237.009,A 0.000,B 0.000,C 90.000,E1 37.523} C_DIS
LIN {X -0.131,Y -595.219,Z 1237.003,A 0.000,B 0.000,C 90.000,E1 36.503} C_DIS
LIN {X 0.195,Y -594.114,Z 1236.998,A 0.000,B 0.000,C 90.000,E1 35.678} C_DIS
LIN {X 0.247,Y -592.403,Z 1236.992,A 0.000,B 0.000,C 90.000,E1 34.612} C_DIS
LIN {X 0.058,Y -590.916,Z 1236.988,A 0.000,B 0.000,C 90.000,E1 33.833} C_DIS
LIN {X 0.141,Y -589.780,Z 1236.985,A 0.000,B 0.000,C 90.000,E1 33.293} C_DIS
LIN {X 0.286,Y -587.031,Z 1236.979,A 0.000,B 0.000,C 90.000,E1 32.212} C_DIS
LIN {X -0.281,Y -584.670,Z 1236.975,A 0.000,B 0.000,C 90.000,E1 31.465} C_DIS
LIN {X -0.371,Y -581.895,Z 1236.970,A 0.000,B 0.000,C 90.000,E1 30.669} C_DIS
LIN {X 0.154,Y -579.850,Z 1236.967,A 0.000,B 0.000,C 90.000,E1 30.079} C_DIS
LIN {X 0.017,Y -576.306,Z 1236.963,A 0.000,B 0.000,C 90.000,E1 29.283} C_DIS
LIN {X 0.072,Y -574.417,Z 1236.960,A 0.000,B 0.000,C 90.000,E1 28.871} C_DIS
LIN {X 0.282,Y -569.470,Z 1236.955,A 0.000,B 0.000,C 90.000,E1 27.897} C_DIS
LIN {X -0.154,Y -565.567,Z 1236.951,A 0.000,B 0.000,C 90.000,E1 27.257} C_DIS
LIN {X 0.041,Y -560.451,Z 1236.947,A 0.000,B 0.000,C 90.000,E1 26.411} C_DIS
LIN {X 0.243,Y -557.650,Z 1236.944,A 0.000,B 0.000,C 90.000,E1 25.976} C_DIS
LIN {X 0.183,Y -551.870,Z 1236.940,A 0.000,B 0.000,C 90.000,E1 25.155} C_DIS
LIN {X 0.121,Y -546.442,Z 1236.936,A 0.000,B 0.000,C 90.000,E1 24.463} C_DIS
LIN {X -0.244,Y -543.040,Z 1236.934,A 0.000,B 0.000,C 90.000,E1 24.079} C_DIS
LIN {X 0.193,Y -533.109,Z 1236.927,A 0.000,B 0.000,C 90.000,E1 22.898} C_DIS
LIN {X 0.121,Y -527.912,Z 1236.924,A 0.000,B 0.000,C 90.000,E1 22.333} C_DIS
LIN {X 0.156,Y -518.656,Z 1236.919,A 0.000,B 0.000,C 90.000,E1 21.354} C_DIS
LIN {X -0.144,Y -509.172,Z 1236.913,A 0.000,B 0.000,C 90.000,E1 20.429} C_DIS
LIN {X -0.069,Y -497.882,Z 1236.907,A 0.000,B 0.000,C 90.000,E1 19.322} C_DIS
LIN {X 0.070,Y -487.659,Z 1236.902,A 0.000,B 0.000,C 90.000,E1 18.362} C_DIS
LIN {X 0.160,Y -480.328,Z 1236.898,A 0.000,B 0.000,C 90.000,E1 17.692} C_DIS
LIN {X -0.016,Y -465.932,Z 1236.891,A 0.000,B 0.000,C 90.000,E1 16.441} C_DIS
LIN {X 0.086,Y -444.036,Z 1236.880,A 0.000,B 0.000,C 90.000,E1 14.426} C_DIS
LIN {X -0.023,Y -425.326,Z 1236.870,A 0.000,B 0.000,C 90.000,E1 12.591} C_DIS
LIN {X -0.112,Y -403.997,Z 1236.857,A 0.000,B 0.000,C 90.000,E1 10.254} C_DIS
LIN {X 0.127,Y -399.903,Z 1236.854,A 0.000,B 0.000,C 90.000,E1 9.726} C_DIS
LIN {X 0.129,Y -395.849,Z 1236.851,A 0.000,B 0.000,C 90.000,E1 9.151} C_DIS
LIN {X -0.123,Y -394.216,Z 1236.849,A 0.000,B 0.000,C 90.000,E1 8.803} C_DIS
LIN {X -0.161,Y -394.207,Z 1236.849,A 0.000,B 0.000,C 90.000,E1 8.803} C_DIS
LIN {X 0.004,Y -394.134,Z 1236.848,A 0.000,B 0.000,C 90.000,E1 8.624} C_DIS
LIN {X -0.033,Y -394.135,Z 1236.848,A 0.000,B 0.000,C 90.000,E1 8.624} C_DIS
LIN {X 0.037,Y -396.432,Z 1236.845,A 0.000,B 0.000,C 90.000,E1 8.106} C_DIS
LIN {X -0.086,Y -398.558,Z 1236.844,A 0.000,B 0.000,C 90.000,E1 7.871} C_DIS
LIN {X 0.076,Y -401.188,Z 1236.842,A 0.000,B 0.000,C 90.000,E1 7.587} C_DIS
LIN {X -0.019,Y -408.232,Z 1236.839,A 0.000,B 0.000,C 90.000,E1 7.068} C_DIS
LIN {X 0.007,Y -414.743,Z 1236.837,A 0.000,B 0.000,C 90.000,E1 6.606} C_DIS
LIN {X 0.089,Y -425.581,Z 1236.832,A 0.000,B 0.000,C 90.000,E1 5.796} C_DIS
LIN {X -0.029,Y -431.899,Z 1236.830,A 0.000,B 0.000,C 90.000,E1 5.334} C_DIS
LIN {X -0.098,Y -444.478,Z 1236.824,A 0.000,B 0.000,C 90.000,E1 4.359} C_DIS
LIN {X -0.059,Y -456.788,Z 1236.819,A 0.000,B 0.000,C 90.000,E1 3.383} C_DIS
LIN {X 0.155,Y -462.865,Z 1236.816,A 0.000,B 0.000,C 90.000,E1 2.865} C_DIS
LIN {X -0.196,Y -468.933,Z 1236.813,A 0.000,B 0.000,C 90.000,E1 2.407} C_DIS
LIN {X -0.061,Y -473.350,Z 1236.811,A 0.000,B 0.000,C 90.000,E1 2.007} C_DIS
LIN {X -0.138,Y -479.096,Z 1236.808,A 0.000,B 0.000,C 90.000,E1 1.489} C_DIS
LIN {X 0.030,Y -484.689,Z 1236.805,A 0.000,B 0.000,C 90.000,E1 0.917} C_DIS
LIN {X -0.064,Y -491.166,Z 1236.801,A 0.000,B 0.000,C 90.000,E1 0.229} C_DIS
LIN {X 0.167,Y -497.428,Z 1236.797,A 0.000,B 0.000,C 90.000,E1 359.484} C_DIS
LIN {X 0.092,Y -503.378,Z 1236.793,A 0.000,B 0.000,C 90.000,E1 358.740} C_DIS
LIN {X 0.205,Y -508.789,Z 1236.789,A 0.000,B 0.000,C 90.000,E1 357.993} C_DIS
LIN {X 0.231,Y -513.881,Z 1236.785,A 0.000,B 0.000,C 90.000,E1 357.249} C_DIS
LIN {X -0.191,Y -518.620,Z 1236.781,A 0.000,B 0.000,C 90.000,E1 356.560} C_DIS
LIN {X 0.201,Y -522.162,Z 1236.778,A 0.000,B 0.000,C 90.000,E1 355.931} C_DIS
LIN {X 0.135,Y -525.472,Z 1236.774,A 0.000,B 0.000,C 90.000,E1 355.355} C_DIS
LIN {X -0.189,Y -529.220,Z 1236.770,A 0.000,B 0.000,C 90.000,E1 354.666} C_DIS
LIN {X 0.101,Y -532.631,Z 1236.766,A 0.000,B 0.000,C 90.000,E1 353.913} C_DIS
LIN {X 0.115,Y -535.186,Z 1236.763,A 0.000,B 0.000,C 90.000,E1 353.337} C_DIS
LIN {X 0.143,Y -537.556,Z 1236.760,A 0.000,B 0.000,C 90.000,E1 352.761} C_DIS
LIN {X 0.250,Y -540.771,Z 1236.755,A 0.000,B 0.000,C 90.000,E1 351.894} C_DIS
LIN {X -0.148,Y -543.743,Z 1236.750,A 0.000,B 0.000,C 90.000,E1 351.084} C_DIS
LIN {X 0.020,Y -545.585,Z 1236.747,A 0.000,B 0.000,C 90.000,E1 350.500} C_DIS
LIN {X -0.233,Y -548.870,Z 1236.741,A 0.000,B 0.000,C 90.000,E1 349.398} C_DIS
LIN {X 0.085,Y -551.165,Z 1236.736,A 0.000,B 0.000,C 90.000,E1 348.522} C_DIS
LIN {X 0.010,Y -553.906,Z 1236.730,A 0.000,B 0.000,C 90.000,E1 347.409} C_DIS
LIN {X -0.032,Y -556.396,Z 1236.724,A 0.000,B 0.000,C 90.000,E1 346.297} C_DIS
LIN {X 0.090,Y -558.615,Z 1236.718,A 0.000,B 0.000,C 90.000,E1 345.172} C_DIS
LIN {X -0.295,Y -560.669,Z 1236.712,A 0.000,B 0.000,C 90.000,E1 344.102} C_DIS
LIN {X 0.046,Y -562.424,Z 1236.705,A 0.000,B 0.000,C 90.000,E1 342.960} C_DIS
LIN {X -0.119,Y -563.935,Z 1236.699,A 0.000,B 0.000,C 90.000,E1 341.873} C_DIS
LIN {X 0.272,Y -565.217,Z 1236.693,A 0.000,B 0.000,C 90.000,E1 340.732} C_DIS
LIN {X 0.003,Y -565.879,Z 1236.689,A 0.000,B 0.000,C 90.000,E1 339.934} C_DIS
LIN {X -0.060,Y -566.234,Z 1236.686,A 0.000,B 0.000,C 90.000,E1 339.390} C_DIS
LIN {X 0.209,Y -566.471,Z 1236.681,A 0.000,B 0.000,C 90.000,E1 338.539} C_DIS
LIN {X -0.174,Y -566.513,Z 1236.678,A 0.000,B 0.000,C 90.000,E1 338.028} C_DIS
LIN {X 0.093,Y -566.251,Z 1236.673,A 0.000,B 0.000,C 90.000,E1 337.177} C_DIS
LIN {X 0.238,Y -565.914,Z 1236.670,A 0.000,B 0.000,C 90.000,E1 336.613} C_DIS
LIN {X 0.196,Y -565.033,Z 1236.666,A 0.000,B 0.000,C 90.000,E1 335.793} C_DIS
LIN {X 0.146,Y -563.912,Z 1236.661,A 0.000,B 0.000,C 90.000,E1 334.973} C_DIS
LIN {X -0.110,Y -561.838,Z 1236.655,A 0.000,B 0.000,C 90.000,E1 333.896} C_DIS
LIN {X -0.144,Y -559.288,Z 1236.649,A 0.000,B 0.000,C 90.000,E1 332.794} C_DIS
LIN {X -0.055,Y -557.570,Z 1236.646,A 0.000,B 0.000,C 90.000,E1 332.231} C_DIS
LIN {X 0.279,Y -555.795,Z 1236.643,A 0.000,B 0.000,C 90.000,E1 331.641} C_DIS
LIN {X -0.106,Y -552.460,Z 1236.638,A 0.000,B 0.000,C 90.000,E1 330.845} C_DIS
LIN {X 0.190,Y -549.877,Z 1236.635,A 0.000,B 0.000,C 90.000,E1 330.255} C_DIS
LIN {X -0.132,Y -546.316,Z 1236.631,A 0.000,B 0.000,C 90.000,E1 329.587} C_DIS
LIN {X 0.113,Y -543.131,Z 1236.628,A 0.000,B 0.000,C 90.000,E1 328.997} C_DIS
LIN {X -0.265,Y -538.565,Z 1236.624,A 0.000,B 0.000,C 90.000,E1 328.329} C_DIS
LIN {X 0.056,Y -533.669,Z 1236.620,A 0.000,B 0.000,C 90.000,E1 327.582} C_DIS
LIN {X 0.171,Y -527.426,Z 1236.615,A 0.000,B 0.000,C 90.000,E1 326.707} C_DIS
LIN {X -0.091,Y -517.650,Z 1236.608,A 0.000,B 0.000,C 90.000,E1 325.435} C_DIS
LIN {X 0.095,Y -514.607,Z 1236.605,A 0.000,B 0.000,C 90.000,E1 324.975} C_DIS
LIN {X -0.159,Y -511.962,Z 1236.603,A 0.000,B 0.000,C 90.000,E1 324.562} C_DIS
LIN {X -0.160,Y -509.626,Z 1236.600,A 0.000,B 0.000,C 90.000,E1 324.069} C_DIS
LIN {X 0.054,Y -508.682,Z 1236.599,A 0.000,B 0.000,C 90.000,E1 323.749} C_DIS
LIN {X 0.279,Y -507.167,Z 1236.595,A 0.000,B 0.000,C 90.000,E1 323.130} C_DIS
LIN {X -0.015,Y -505.952,Z 1236.590,A 0.000,B 0.000,C 90.000,E1 322.271} C_DIS
LIN {X -0.009,Y -505.452,Z 1236.585,A 0.000,B 0.000,C 90.000,E1 321.376} C_DIS
LIN {X 0.014,Y -506.557,Z 1236.571,A 0.000,B 0.000,C 90.000,E1 318.690} C_DIS
LIN {X -0.232,Y -507.181,Z 1236.562,A 0.000,B 0.000,C 90.000,E1 317.229} C_DIS
LIN {X -0.124,Y -507.696,Z 1236.554,A 0.000,B 0.000,C 90.000,E1 315.729} C_DIS
LIN {X -0.132,Y -508.290,Z 1236.544,A 0.000,B 0.000,C 90.000,E1 313.947} C_DIS
LIN {X 0.129,Y -509.025,Z 1236.533,A 0.000,B 0.000,C 90.000,E1 311.838} C_DIS
LIN {X 0.020,Y -509.489,Z 1236.526,A 0.000,B 0.000,C 90.000,E1 310.663} C_DIS
LIN {X -0.122,Y -510.001,Z 1236.518,A 0.000,B 0.000,C 90.000,E1 309.197} C_DIS
LIN {X -0.249,Y -510.416,Z 1236.510,A 0.000,B 0.000,C 90.000,E1 307.729} C_DIS
LIN {X 0.032,Y -510.851,Z 1236.501,A 0.000,B 0.000,C 90.000,E1 306.217} C_DIS
LIN {X 0.018,Y -511.206,Z 1236.493,A 0.000,B 0.000,C 90.000,E1 304.739} C_DIS
LIN {X 0.146,Y -511.550,Z 1236.485,A 0.000,B 0.000,C 90.000,E1 303.245} C_DIS
LIN {X -0.145,Y -511.691,Z 1236.477,A 0.000,B 0.000,C 90.000,E1 301.799} C_DIS
LIN {X 0.072,Y -511.825,Z 1236.467,A 0.000,B 0.000,C 90.000,E1 300.001} C_DIS
LIN {X -0.059,Y -511.873,Z 1236.458,A 0.000,B 0.000,C 90.000,E1 298.537} C_DIS
LIN {X 0.009,Y -511.857,Z 1236.450,A 0.000,B 0.000,C 90.000,E1 297.052} C_DIS
LIN {X -0.065,Y -511.922,Z 1236.437,A 0.000,B 0.000,C 90.000,E1 294.695} C_DIS
LIN {X 0.034,Y -512.066,Z 1236.429,A 0.000,B 0.000,C 90.000,E1 293.206} C_DIS
LIN {X -0.089,Y -511.886,Z 1236.424,A 0.000,B 0.000,C 90.000,E1 292.333} C_DIS
LIN {X 0.008,Y -511.420,Z 1236.416,A 0.000,B 0.000,C 90.000,E1 290.844} C_DIS
LIN {X -0.154,Y -510.577,Z 1236.406,A 0.000,B 0.000,C 90.000,E1 289.087} C_DIS
LIN {X 0.154,Y -509.954,Z 1236.396,A 0.000,B 0.000,C 90.000,E1 287.275} C_DIS
LIN {X 0.242,Y -508.975,Z 1236.385,A 0.000,B 0.000,C 90.000,E1 285.190} C_DIS
LIN {X 0.188,Y -508.259,Z 1236.378,A 0.000,B 0.000,C 90.000,E1 284.008} C_DIS
LIN {X 0.217,Y -507.947,Z 1236.375,A 0.000,B 0.000,C 90.000,E1 283.411} C_DIS
LIN {X -0.063,Y -506.737,Z 1236.365,A 0.000,B 0.000,C 90.000,E1 281.658} C_DIS
LIN {X 0.210,Y -504.182,Z 1236.345,A 0.000,B 0.000,C 90.000,E1 278.049} C_DIS
LIN {X -0.242,Y -503.250,Z 1236.337,A 0.000,B 0.000,C 90.000,E1 276.606} C_DIS
LIN {X 0.208,Y -502.342,Z 1236.327,A 0.000,B 0.000,C 90.000,E1 274.759} C_DIS
LIN {X 0.135,Y -501.491,Z 1236.318,A 0.000,B 0.000,C 90.000,E1 273.269} C_DIS
LIN {X -0.050,Y -500.205,Z 1236.308,A 0.000,B 0.000,C 90.000,E1 271.489} C_DIS
LIN {X 0.077,Y -498.652,Z 1236.297,A 0.000,B 0.000,C 90.000,E1 269.370} C_DIS
LIN {X -0.179,Y -498.253,Z 1236.293,A 0.000,B 0.000,C 90.000,E1 268.797} C_DIS
LIN {X 0.039,Y -497.200,Z 1236.283,A 0.000,B 0.000,C 90.000,E1 266.963} C_DIS
LIN {X 0.045,Y -496.525,Z 1236.276,A 0.000,B 0.000,C 90.000,E1 265.755} C_DIS
LIN {X 0.050,Y -495.829,Z 1236.270,A 0.000,B 0.000,C 90.000,E1 264.546} C_DIS
LIN {X -0.211,Y -494.536,Z 1236.260,A 0.000,B 0.000,C 90.000,E1 262.761} C_DIS
LIN {X 0.209,Y -493.171,Z 1236.251,A 0.000,B 0.000,C 90.000,E1 261.197} C_DIS
LIN {X -0.199,Y -490.806,Z 1236.238,A 0.000,B 0.000,C 90.000,E1 258.814} C_DIS
LIN {X 0.104,Y -489.219,Z 1236.226,A 0.000,B 0.000,C 90.000,E1 256.645} C_DIS
LIN {X -0.001,Y -487.912,Z 1236.214,A 0.000,B 0.000,C 90.000,E1 254.519} C_DIS
LIN {X 0.134,Y -486.427,Z 1236.200,A 0.000,B 0.000,C 90.000,E1 252.054} C_DIS
LIN {X -0.110,Y -485.724,Z 1236.192,A 0.000,B 0.000,C 90.000,E1 250.550} C_DIS
LIN {X -0.215,Y -484.951,Z 1236.183,A 0.000,B 0.000,C 90.000,E1 249.028} C_DIS
LIN {X -0.162,Y -484.124,Z 1236.175,A 0.000,B 0.000,C 90.000,E1 247.486} C_DIS
LIN {X 0.062,Y -483.106,Z 1236.166,A 0.000,B 0.000,C 90.000,E1 245.921} C_DIS
LIN {X 0.032,Y -481.691,Z 1236.156,A 0.000,B 0.000,C 90.000,E1 244.076} C_DIS
LIN {X -0.016,Y -480.540,Z 1236.147,A 0.000,B 0.000,C 90.000,E1 242.538} C_DIS
LIN {X 0.106,Y -478.905,Z 1236.137,A 0.000,B 0.000,C 90.000,E1 240.667} C_DIS
LIN {X 0.043,Y -477.364,Z 1236.129,A 0.000,B 0.000,C 90.000,E1 239.125} C_DIS
LIN {X 0.167,Y -476.092,Z 1236.122,A 0.000,B 0.000,C 90.000,E1 237.867} C_DIS
LIN {X 0.090,Y -474.273,Z 1236.111,A 0.000,B 0.000,C 90.000,E1 236.008} C_DIS
LIN {X 0.028,Y -472.202,Z 1236.099,A 0.000,B 0.000,C 90.000,E1 233.829} C_DIS
LIN {X -0.246,Y -471.343,Z 1236.094,A 0.000,B 0.000,C 90.000,E1 232.924} C_DIS
LIN {X 0.030,Y -469.652,Z 1236.083,A 0.000,B 0.000,C 90.000,E1 231.009} C_DIS
LIN {X -0.160,Y -468.310,Z 1236.075,A 0.000,B 0.000,C 90.000,E1 229.461} C_DIS
LIN {X -0.010,Y -466.822,Z 1236.064,A 0.000,B 0.000,C 90.000,E1 227.553} C_DIS
LIN {X 0.143,Y -465.218,Z 1236.052,A 0.000,B 0.000,C 90.000,E1 225.324} C_DIS
LIN {X -0.076,Y -463.771,Z 1236.031,A 0.000,B 0.000,C 90.000,E1 221.553} C_DIS
LIN {X 0.048,Y -465.188,Z 1235.997,A 0.000,B 0.000,C 90.000,E1 215.518} C_DIS
LIN {X -0.068,Y -468.742,Z 1235.971,A 0.000,B 0.000,C 90.000,E1 210.797} C_DIS
LIN {X 0.056,Y -472.191,Z 1235.954,A 0.000,B 0.000,C 90.000,E1 207.641} C_DIS
LIN {X -0.031,Y -474.924,Z 1235.942,A 0.000,B 0.000,C 90.000,E1 205.463} C_DIS
LIN {X 0.125,Y -479.982,Z 1235.922,A 0.000,B 0.000,C 90.000,E1 202.025} C_DIS
LIN {X -0.190,Y -486.782,Z 1235.902,A 0.000,B 0.000,C 90.000,E1 198.362} C_DIS
LIN {X -0.138,Y -492.925,Z 1235.887,A 0.000,B 0.000,C 90.000,E1 195.607} C_DIS
LIN {X -0.003,Y -497.324,Z 1235.877,A 0.000,B 0.000,C 90.000,E1 193.772} C_DIS
LIN {X 0.121,Y -501.890,Z 1235.867,A 0.000,B 0.000,C 90.000,E1 191.951} C_DIS
LIN {X 0.094,Y -508.999,Z 1235.852,A 0.000,B 0.000,C 90.000,E1 189.265} C_DIS
LIN {X -0.190,Y -513.123,Z 1235.843,A 0.000,B 0.000,C 90.000,E1 187.814} C_DIS
LIN {X 0.038,Y -517.099,Z 1235.835,A 0.000,B 0.000,C 90.000,E1 186.315} C_DIS
LIN {X -0.240,Y -521.896,Z 1235.825,A 0.000,B 0.000,C 90.000,E1 184.588} C_DIS
LIN {X 0.030,Y -527.416,Z 1235.814,A 0.000,B 0.000,C 90.000,E1 182.522} C_DIS
LIN {X -0.077,Y -531.315,Z 1235.806,A 0.000,B 0.000,C 90.000,E1 181.088} C_DIS
LIN {X -0.122,Y -534.403,Z 1235.800,A 0.000,B 0.000,C 90.000,E1 179.943} C_DIS
LIN {X -0.117,Y -538.151,Z 1235.792,A 0.000,B 0.000,C 90.000,E1 178.511} C_DIS
LIN {X -0.033,Y -541.709,Z 1235.784,A 0.000,B 0.000,C 90.000,E1 177.078} C_DIS
LIN {X 0.123,Y -544.438,Z 1235.777,A 0.000,B 0.000,C 90.000,E1 175.927} C_DIS
LIN {X -0.147,Y -548.403,Z 1235.768,A 0.000,B 0.000,C 90.000,E1 174.261} C_DIS
LIN {X 0.215,Y -551.479,Z 1235.760,A 0.000,B 0.000,C 90.000,E1 172.818} C_DIS
LIN {X 0.207,Y -555.128,Z 1235.751,A 0.000,B 0.000,C 90.000,E1 171.141} C_DIS
LIN {X -0.187,Y -558.608,Z 1235.742,A 0.000,B 0.000,C 90.000,E1 169.511} C_DIS
LIN {X -0.119,Y -561.425,Z 1235.734,A 0.000,B 0.000,C 90.000,E1 168.117} C_DIS
LIN {X -0.156,Y -564.856,Z 1235.725,A 0.000,B 0.000,C 90.000,E1 166.464} C_DIS
LIN {X 0.060,Y -568.961,Z 1235.714,A 0.000,B 0.000,C 90.000,E1 164.519} C_DIS
LIN {X 0.132,Y -576.564,Z 1235.697,A 0.000,B 0.000,C 90.000,E1 161.511} C_DIS
LIN {X -0.185,Y -580.894,Z 1235.690,A 0.000,B 0.000,C 90.000,E1 160.188} C_DIS
LIN {X -0.031,Y -585.800,Z 1235.682,A 0.000,B 0.000,C 90.000,E1 158.827} C_DIS
LIN {X -0.107,Y -595.889,Z 1235.669,A 0.000,B 0.000,C 90.000,E1 156.433} C_DIS
LIN {X 0.012,Y -601.598,Z 1235.662,A 0.000,B 0.000,C 90.000,E1 155.101} C_DIS
LIN {X 0.239,Y -607.325,Z 1235.654,A 0.000,B 0.000,C 90.000,E1 153.768} C_DIS
LIN {X 0.015,Y -612.755,Z 1235.647,A 0.000,B 0.000,C 90.000,E1 152.487} C_DIS
LIN {X 0.168,Y -617.906,Z 1235.640,A 0.000,B 0.000,C 90.000,E1 151.179} C_DIS
LIN {X -0.133,Y -623.833,Z 1235.631,A 0.000,B 0.000,C 90.000,E1 149.665} C_DIS
LIN {X 0.190,Y -627.814,Z 1235.626,A 0.000,B 0.000,C 90.000,E1 148.614} C_DIS
LIN {X 0.363,Y -631.580,Z 1235.620,A 0.000,B 0.000,C 90.000,E1 147.582} C_DIS
LIN {X 0.090,Y -636.117,Z 1235.613,A 0.000,B 0.000,C 90.000,E1 146.342} C_DIS
LIN {X -0.112,Y -640.325,Z 1235.606,A 0.000,B 0.000,C 90.000,E1 145.102} C_DIS
LIN {X -0.207,Y -641.979,Z 1235.603,A 0.000,B 0.000,C 90.000,E1 144.609} C_DIS
LIN {X 0.052,Y -645.612,Z 1235.596,A 0.000,B 0.000,C 90.000,E1 143.336} C_DIS
LIN {X -0.148,Y -648.932,Z 1235.589,A 0.000,B 0.000,C 90.000,E1 142.110} C_DIS
LIN {X -0.301,Y -652.028,Z 1235.583,A 0.000,B 0.000,C 90.000,E1 140.884} C_DIS
LIN {X 0.003,Y -654.962,Z 1235.576,A 0.000,B 0.000,C 90.000,E1 139.622} C_DIS
LIN {X -0.145,Y -657.872,Z 1235.569,A 0.000,B 0.000,C 90.000,E1 138.405} C_DIS
LIN {X 0.223,Y -660.177,Z 1235.563,A 0.000,B 0.000,C 90.000,E1 137.391} C_DIS
LIN {X -0.354,Y -664.131,Z 1235.554,A 0.000,B 0.000,C 90.000,E1 135.729} C_DIS
LIN {X -0.375,Y -669.028,Z 1235.543,A 0.000,B 0.000,C 90.000,E1 133.785} C_DIS
LIN {X -0.263,Y -673.387,Z 1235.534,A 0.000,B 0.000,C 90.000,E1 132.081} C_DIS
LIN {X -0.079,Y -677.115,Z 1235.526,A 0.000,B 0.000,C 90.000,E1 130.620} C_DIS
LIN {X 0.135,Y -680.196,Z 1235.519,A 0.000,B 0.000,C 90.000,E1 129.402} C_DIS
LIN {X 0.106,Y -683.859,Z 1235.511,A 0.000,B 0.000,C 90.000,E1 127.971} C_DIS
LIN {X -0.388,Y -687.489,Z 1235.503,A 0.000,B 0.000,C 90.000,E1 126.583} C_DIS
LIN {X -0.137,Y -689.202,Z 1235.499,A 0.000,B 0.000,C 90.000,E1 125.851} C_DIS
LIN {X 0.170,Y -692.398,Z 1235.491,A 0.000,B 0.000,C 90.000,E1 124.405} C_DIS
LIN {X -0.031,Y -695.551,Z 1235.483,A 0.000,B 0.000,C 90.000,E1 123.007} C_DIS
LIN {X 0.097,Y -697.001,Z 1235.479,A 0.000,B 0.000,C 90.000,E1 122.291} C_DIS
LIN {X 0.194,Y -699.724,Z 1235.472,A 0.000,B 0.000,C 90.000,E1 120.875} C_DIS
LIN {X 0.048,Y -701.472,Z 1235.466,A 0.000,B 0.000,C 90.000,E1 119.951} C_DIS
LIN {X -0.075,Y -703.053,Z 1235.461,A 0.000,B 0.000,C 90.000,E1 119.027} C_DIS
LIN {X -0.184,Y -704.389,Z 1235.456,A 0.000,B 0.000,C 90.000,E1 118.103} C_DIS
LIN {X 0.340,Y -705.275,Z 1235.451,A 0.000,B 0.000,C 90.000,E1 117.129} C_DIS
LIN {X -0.075,Y -705.881,Z 1235.446,A 0.000,B 0.000,C 90.000,E1 116.232} C_DIS
LIN {X -0.141,Y -706.002,Z 1235.442,A 0.000,B 0.000,C 90.000,E1 115.540} C_DIS
LIN {X -0.195,Y -705.895,Z 1235.439,A 0.000,B 0.000,C 90.000,E1 115.079} C_DIS
LIN {X 0.090,Y -705.541,Z 1235.437,A 0.000,B 0.000,C 90.000,E1 114.591} C_DIS
LIN {X 0.025,Y -704.779,Z 1235.434,A 0.000,B 0.000,C 90.000,E1 114.131} C_DIS
LIN {X 0.024,Y -704.265,Z 1235.433,A 0.000,B 0.000,C 90.000,E1 113.898} C_DIS
LIN {X -0.194,Y -701.560,Z 1235.430,A 0.000,B 0.000,C 90.000,E1 113.334} C_DIS
LIN {X -0.056,Y -700.687,Z 1235.429,A 0.000,B 0.000,C 90.000,E1 113.206} C_DIS
LIN {X -0.331,Y -695.836,Z 1235.426,A 0.000,B 0.000,C 90.000,E1 112.770} C_DIS
LIN {X -0.171,Y -694.255,Z 1235.426,A 0.000,B 0.000,C 90.000,E1 112.642} C_DIS
LIN {X -0.012,Y -691.473,Z 1235.425,A 0.000,B 0.000,C 90.000,E1 112.514} C_DIS
LIN {X 0.013,Y -685.813,Z 1235.424,A 0.000,B 0.000,C 90.000,E1 112.333} C_DIS
LIN {X 0.026,Y -679.669,Z 1235.424,A 0.000,B 0.000,C 90.000,E1 112.280} C_DIS
LIN {X -0.179,Y -676.996,Z 1235.424,A 0.000,B 0.000,C 90.000,E1 112.280} C_DIS
LIN {X -0.212,Y -619.525,Z 1235.424,A 0.000,B 0.000,C 90.000,E1 112.280} C_DIS
LIN {X 0.246,Y -616.043,Z 1235.422,A 0.000,B 0.000,C 90.000,E1 112.025} C_DIS
LIN {X -0.029,Y -614.093,Z 1235.421,A 0.000,B 0.000,C 90.000,E1 111.844} C_DIS
LIN {X -0.072,Y -614.076,Z 1235.421,A 0.000,B 0.000,C 90.000,E1 111.844} C_DIS
LIN {X 0.105,Y -613.609,Z 1235.420,A 0.000,B 0.000,C 90.000,E1 111.663} C_DIS
LIN {X 0.062,Y -613.609,Z 1235.420,A 0.000,B 0.000,C 90.000,E1 111.663} C_DIS
LIN {X -0.008,Y -614.361,Z 1235.419,A 0.000,B 0.000,C 90.000,E1 111.354} C_DIS
LIN {X -0.120,Y -615.589,Z 1235.417,A 0.000,B 0.000,C 90.000,E1 111.046} C_DIS
LIN {X -0.191,Y -618.131,Z 1235.414,A 0.000,B 0.000,C 90.000,E1 110.536} C_DIS
LIN {X -0.124,Y -621.819,Z 1235.410,A 0.000,B 0.000,C 90.000,E1 109.758} C_DIS
LIN {X 0.193,Y -625.016,Z 1235.406,A 0.000,B 0.000,C 90.000,E1 108.960} C_DIS
LIN {X 0.134,Y -629.147,Z 1235.400,A 0.000,B 0.000,C 90.000,E1 107.946} C_DIS
LIN {X 0.138,Y -634.880,Z 1235.393,A 0.000,B 0.000,C 90.000,E1 106.677} C_DIS
LIN {X -0.045,Y -636.031,Z 1235.391,A 0.000,B 0.000,C 90.000,E1 106.441} C_DIS
LIN {X -0.224,Y -638.135,Z 1235.389,A 0.000,B 0.000,C 90.000,E1 105.953} C_DIS
LIN {X 0.217,Y -639.312,Z 1235.387,A 0.000,B 0.000,C 90.000,E1 105.662} C_DIS
LIN {X -0.277,Y -641.952,Z 1235.383,A 0.000,B 0.000,C 90.000,E1 104.954} C_DIS
LIN {X 0.032,Y -643.523,Z 1235.380,A 0.000,B 0.000,C 90.000,E1 104.426} C_DIS
LIN {X 0.362,Y -645.478,Z 1235.376,A 0.000,B 0.000,C 90.000,E1 103.647} C_DIS
LIN {X 0.070,Y -646.442,Z 1235.373,A 0.000,B 0.000,C 90.000,E1 103.175} C_DIS
LIN {X -0.218,Y -647.132,Z 1235.370,A 0.000,B 0.000,C 90.000,E1 102.703} C_DIS
LIN {X -0.008,Y -647.556,Z 1235.368,A 0.000,B 0.000,C 90.000,E1 102.187} C_DIS
LIN {X -0.147,Y -647.639,Z 1235.366,A 0.000,B 0.000,C 90.000,E1 101.951} C_DIS
LIN {X 0.208,Y -647.502,Z 1235.364,A 0.000,B 0.000,C 90.000,E1 101.422} C_DIS
LIN {X -0.074,Y -646.869,Z 1235.361,A 0.000,B 0.000,C 90.000,E1 100.950} C_DIS
LIN {X 0.153,Y -645.906,Z 1235.358,A 0.000,B 0.000,C 90.000,E1 100.433} C_DIS
LIN {X 0.007,Y -645.345,Z 1235.357,A 0.000,B 0.000,C 90.000,E1 100.197} C_DIS
LIN {X 0.341,Y -643.951,Z 1235.354,A 0.000,B 0.000,C 90.000,E1 99.670} C_DIS
LIN {X -0.078,Y -642.156,Z 1235.351,A 0.000,B 0.000,C 90.000,E1 99.208} C_DIS
LIN {X -0.039,Y -638.705,Z 1235.347,A 0.000,B 0.000,C 90.000,E1 98.454} C_DIS
LIN {X 0.148,Y -635.999,Z 1235.344,A 0.000,B 0.000,C 90.000,E1 97.936} C_DIS
LIN {X -0.230,Y -632.961,Z 1235.341,A 0.000,B 0.000,C 90.000,E1 97.466} C_DIS
LIN {X -0.231,Y -628.301,Z 1235.338,A 0.000,B 0.000,C 90.000,E1 96.834} C_DIS
LIN {X 0.032,Y -625.347,Z 1235.336,A 0.000,B 0.000,C 90.000,E1 96.429} C_DIS
LIN {X -0.105,Y -617.989,Z 1235.332,A 0.000,B 0.000,C 90.000,E1 95.682} C_DIS
LIN {X 0.216,Y -612.539,Z 1235.329,A 0.000,B 0.000,C 90.000,E1 95.163} C_DIS
LIN {X 0.213,Y -608.250,Z 1235.327,A 0.000,B 0.000,C 90.000,E1 94.821} C_DIS
LIN {X -0.128,Y -602.283,Z 1235.324,A 0.000,B 0.000,C 90.000,E1 94.416} C_DIS
LIN {X 0.191,Y -597.645,Z 1235.323,A 0.000,B 0.000,C 90.000,E1 94.073} C_DIS
LIN {X -0.026,Y -589.814,Z 1235.320,A 0.000,B 0.000,C 90.000,E1 93.612} C_DIS
LIN {X -0.195,Y -583.207,Z 1235.318,A 0.000,B 0.000,C 90.000,E1 93.269} C_DIS
LIN {X -0.109,Y -579.688,Z 1235.317,A 0.000,B 0.000,C 90.000,E1 93.094} C_DIS
LIN {X 0.238,Y -571.011,Z 1235.315,A 0.000,B 0.000,C 90.000,E1 92.694} C_DIS
LIN {X -0.154,Y -567.214,Z 1235.314,A 0.000,B 0.000,C 90.000,E1 92.522} C_DIS
LIN {X -0.196,Y -567.142,Z 1235.314,A 0.000,B 0.000,C 90.000,E1 92.522} C_DIS
LIN {X 0.248,Y -566.162,Z 1235.313,A 0.000,B 0.000,C 90.000,E1 92.293} C_DIS
LIN {X 0.207,Y -566.147,Z 1235.313,A 0.000,B 0.000,C 90.000,E1 92.293} C_DIS
LIN {X -0.102,Y -566.061,Z 1235.312,A 0.000,B 0.000,C 90.000,E1 92.178} C_DIS
LIN {X 0.013,Y -565.660,Z 1235.311,A 0.000,B 0.000,C 90.000,E1 91.892} C_DIS
LIN {X 0.034,Y -566.280,Z 1235.303,A 0.000,B 0.000,C 90.000,E1 90.516} C_DIS
LIN {X 0.171,Y -567.477,Z 1235.294,A 0.000,B 0.000,C 90.000,E1 88.854} C_DIS
LIN {X 0.048,Y -569.143,Z 1235.282,A 0.000,B 0.000,C 90.000,E1 86.674} C_DIS
LIN {X 0.019,Y -571.040,Z 1235.269,A 0.000,B 0.000,C 90.000,E1 84.489} C_DIS
LIN {X -0.213,Y -572.638,Z 1235.260,A 0.000,B 0.000,C 90.000,E1 82.875} C_DIS
LIN {X 0.227,Y -574.228,Z 1235.251,A 0.000,B 0.000,C 90.000,E1 81.197} C_DIS
LIN {X 0.016,Y -575.388,Z 1235.244,A 0.000,B 0.000,C 90.000,E1 79.859} C_DIS
LIN {X -0.179,Y -576.326,Z 1235.236,A 0.000,B 0.000,C 90.000,E1 78.522} C_DIS
LIN {X -0.035,Y -577.402,Z 1235.227,A 0.000,B 0.000,C 90.000,E1 76.881} C_DIS
LIN {X 0.262,Y -578.391,Z 1235.218,A 0.000,B 0.000,C 90.000,E1 75.227} C_DIS
LIN {X 0.176,Y -579.279,Z 1235.209,A 0.000,B 0.000,C 90.000,E1 73.614} C_DIS
LIN {X -0.273,Y -580.058,Z 1235.202,A 0.000,B 0.000,C 90.000,E1 72.308} C_DIS
LIN {X 0.234,Y -581.237,Z 1235.191,A 0.000,B 0.000,C 90.000,E1 70.369} C_DIS
LIN {X -0.161,Y -583.356,Z 1235.173,A 0.000,B 0.000,C 90.000,E1 67.177} C_DIS
LIN {X 0.008,Y -584.987,Z 1235.163,A 0.000,B 0.000,C 90.000,E1 65.281} C_DIS
LIN {X -0.011,Y -587.197,Z 1235.149,A 0.000,B 0.000,C 90.000,E1 62.871} C_DIS
LIN {X -0.017,Y -589.054,Z 1235.139,A 0.000,B 0.000,C 90.000,E1 61.001} C_DIS
LIN {X 0.117,Y -590.148,Z 1235.133,A 0.000,B 0.000,C 90.000,E1 59.921} C_DIS
LIN {X -0.025,Y -591.282,Z 1235.127,A 0.000,B 0.000,C 90.000,E1 58.869} C_DIS
LIN {X 0.152,Y -592.291,Z 1235.121,A 0.000,B 0.000,C 90.000,E1 57.788} C_DIS
LIN {X -0.055,Y -593.792,Z 1235.112,A 0.000,B 0.000,C 90.000,E1 56.215} C_DIS
LIN {X -0.122,Y -594.936,Z 1235.105,A 0.000,B 0.000,C 90.000,E1 54.895} C_DIS
LIN {X 0.049,Y -596.179,Z 1235.096,A 0.000,B 0.000,C 90.000,E1 53.290} C_DIS
LIN {X -0.119,Y -597.633,Z 1235.086,A 0.000,B 0.000,C 90.000,E1 51.457} C_DIS
LIN {X 0.118,Y -598.144,Z 1235.081,A 0.000,B 0.000,C 90.000,E1 50.642} C_DIS
LIN {X -0.013,Y -599.007,Z 1235.071,A 0.000,B 0.000,C 90.000,E1 48.809} C_DIS
LIN {X 0.191,Y -599.596,Z 1235.064,A 0.000,B 0.000,C 90.000,E1 47.472} C_DIS
LIN {X -0.225,Y -599.837,Z 1235.058,A 0.000,B 0.000,C 90.000,E1 46.458} C_DIS
LIN {X -0.006,Y -599.935,Z 1235.051,A 0.000,B 0.000,C 90.000,E1 45.121} C_DIS
LIN {X 0.213,Y -599.765,Z 1235.043,A 0.000,B 0.000,C 90.000,E1 43.785} C_DIS
LIN {X 0.014,Y -599.561,Z 1235.039,A 0.000,B 0.000,C 90.000,E1 43.014} C_DIS
LIN {X 0.219,Y -599.243,Z 1235.035,A 0.000,B 0.000,C 90.000,E1 42.204} C_DIS
LIN {X 0.245,Y -598.720,Z 1235.029,A 0.000,B 0.000,C 90.000,E1 41.148} C_DIS
LIN {X 0.274,Y -597.934,Z 1235.020,A 0.000,B 0.000,C 90.000,E1 39.564} C_DIS
LIN {X -0.330,Y -597.429,Z 1235.016,A 0.000,B 0.000,C 90.000,E1 38.830} C_DIS
LIN {X 0.132,Y -596.389,Z 1235.010,A 0.000,B 0.000,C 90.000,E1 37.729} C_DIS
LIN {X -0.036,Y -594.884,Z 1235.002,A 0.000,B 0.000,C 90.000,E1 36.423} C_DIS
LIN {X 0.285,Y -593.763,Z 1234.998,A 0.000,B 0.000,C 90.000,E1 35.598} C_DIS
LIN {X -0.007,Y -592.011,Z 1234.992,A 0.000,B 0.000,C 90.000,E1 34.565} C_DIS
LIN {X -0.194,Y -590.465,Z 1234.988,A 0.000,B 0.000,C 90.000,E1 33.785} C_DIS
LIN {X 0.088,Y -588.681,Z 1234.983,A 0.000,B 0.000,C 90.000,E1 32.959} C_DIS
LIN {X 0.347,Y -586.573,Z 1234.979,A 0.000,B 0.000,C 90.000,E1 32.133} C_DIS
LIN {X 0.271,Y -584.106,Z 1234.974,A 0.000,B 0.000,C 90.000,E1 31.337} C_DIS
LIN {X 0.310,Y -582.312,Z 1234.971,A 0.000,B 0.000,C 90.000,E1 30.797} C_DIS
LIN {X 0.194,Y -579.187,Z 1234.967,A 0.000,B 0.000,C 90.000,E1 30.001} C_DIS
LIN {X 0.119,Y -576.195,Z 1234.963,A 0.000,B 0.000,C 90.000,E1 29.333} C_DIS
LIN {X -0.185,Y -573.656,Z 1234.960,A 0.000,B 0.000,C 90.000,E1 28.821} C_DIS
LIN {X 0.105,Y -569.374,Z 1234.956,A 0.000,B 0.000,C 90.000,E1 27.975} C_DIS
LIN {X -0.066,Y -565.535,Z 1234.952,A 0.000,B 0.000,C 90.000,E1 27.308} C_DIS
LIN {X -0.126,Y -560.411,Z 1234.947,A 0.000,B 0.000,C 90.000,E1 26.488} C_DIS
LIN {X -0.096,Y -554.896,Z 1234.943,A 0.000,B 0.000,C 90.000,E1 25.668} C_DIS
LIN {X 0.203,Y -550.900,Z 1234.939,A 0.000,B 0.000,C 90.000,E1 25.079} C_DIS
LIN {X 0.017,Y -544.229,Z 1234.935,A 0.000,B 0.000,C 90.000,E1 24.259} C_DIS
LIN {X 0.006,Y -538.350,Z 1234.931,A 0.000,B 0.000,C 90.000,E1 23.567} C_DIS
LIN {X 0.100,Y -530.947,Z 1234.926,A 0.000,B 0.000,C 90.000,E1 22.717} C_DIS
LIN {X -0.096,Y -521.864,Z 1234.921,A 0.000,B 0.000,C 90.000,E1 21.770} C_DIS
LIN {X -0.123,Y -517.834,Z 1234.919,A 0.000,B 0.000,C 90.000,E1 21.354} C_DIS
LIN {X 0.162,Y -508.486,Z 1234.913,A 0.000,B 0.000,C 90.000,E1 20.375} C_DIS
LIN {X 0.122,Y -497.555,Z 1234.907,A 0.000,B 0.000,C 90.000,E1 19.322} C_DIS
LIN {X -0.160,Y -488.791,Z 1234.903,A 0.000,B 0.000,C 90.000,E1 18.544} C_DIS
LIN {X -0.143,Y -479.955,Z 1234.899,A 0.000,B 0.000,C 90.000,E1 17.747} C_DIS
LIN {X -0.098,Y -466.478,Z 1234.892,A 0.000,B 0.000,C 90.000,E1 16.551} C_DIS
LIN {X -0.105,Y -448.804,Z 1234.883,A 0.000,B 0.000,C 90.000,E1 14.954} C_DIS
LIN {X -0.023,Y -427.139,Z 1234.871,A 0.000,B 0.000,C 90.000,E1 12.827} C_DIS
LIN {X 0.049,Y -408.907,Z 1234.860,A 0.000,B 0.000,C 90.000,E1 10.838} C_DIS
LIN {X -0.198,Y -400.614,Z 1234.855,A 0.000,B 0.000,C 90.000,E1 9.905} C_DIS
LIN {X -0.048,Y -397.920,Z 1234.853,A 0.000,B 0.000,C 90.000,E1 9.500} C_DIS
LIN {X -0.062,Y -395.529,Z 1234.851,A 0.000,B 0.000,C 90.000,E1 9.151} C_DIS
LIN {X -0.089,Y -394.120,Z 1234.849,A 0.000,B 0.000,C 90.000,E1 8.803} C_DIS
LIN {X -0.128,Y -394.116,Z 1234.849,A 0.000,B 0.000,C 90.000,E1 8.803} C_DIS
LIN {X 0.114,Y -394.072,Z 1234.848,A 0.000,B 0.000,C 90.000,E1 8.624} C_DIS
LIN {X 0.076,Y -394.071,Z 1234.848,A 0.000,B 0.000,C 90.000,E1 8.624} C_DIS
LIN {X -0.199,Y -396.693,Z 1234.845,A 0.000,B 0.000,C 90.000,E1 8.106} C_DIS
LIN {X 0.096,Y -399.925,Z 1234.843,A 0.000,B 0.000,C 90.000,E1 7.701} C_DIS
LIN {X -0.178,Y -403.834,Z 1234.841,A 0.000,B 0.000,C 90.000,E1 7.409} C_DIS
LIN {X -0.221,Y -414.915,Z 1234.837,A 0.000,B 0.000,C 90.000,E1 6.606} C_DIS
LIN {X 0.105,Y -419.720,Z 1234.835,A 0.000,B 0.000,C 90.000,E1 6.201} C_DIS
LIN {X -0.144,Y -424.337,Z 1234.833,A 0.000,B 0.000,C 90.000,E1 5.910} C_DIS
LIN {X -0.182,Y -431.939,Z 1234.830,A 0.000,B 0.000,C 90.000,E1 5.334} C_DIS
LIN {X 0.137,Y -446.113,Z 1234.823,A 0.000,B 0.000,C 90.000,E1 4.188} C_DIS
LIN {X 0.168,Y -457.054,Z 1234.819,A 0.000,B 0.000,C 90.000,E1 3.326} C_DIS
LIN {X 0.219,Y -466.262,Z 1234.815,A 0.000,B 0.000,C 90.000,E1 2.579} C_DIS
LIN {X -0.157,Y -472.231,Z 1234.812,A 0.000,B 0.000,C 90.000,E1 2.121} C_DIS
LIN {X 0.120,Y -479.355,Z 1234.808,A 0.000,B 0.000,C 90.000,E1 1.432} C_DIS
LIN {X 0.072,Y -484.713,Z 1234.805,A 0.000,B 0.000,C 90.000,E1 0.917} C_DIS
LIN {X -0.209,Y -491.454,Z 1234.801,A 0.000,B 0.000,C 90.000,E1 0.229} C_DIS
LIN {X 0.104,Y -497.643,Z 1234.797,A 0.000,B 0.000,C 90.000,E1 359.484} C_DIS
LIN {X 0.030,Y -503.621,Z 1234.793,A 0.000,B 0.000,C 90.000,E1 358.740} C_DIS
LIN {X 0.022,Y -509.189,Z 1234.789,A 0.000,B 0.000,C 90.000,E1 357.993} C_DIS
LIN {X 0.050,Y -514.334,Z 1234.785,A 0.000,B 0.000,C 90.000,E1 357.249} C_DIS
LIN {X 0.149,Y -519.065,Z 1234.781,A 0.000,B 0.000,C 90.000,E1 356.502} C_DIS
LIN {X 0.061,Y -522.610,Z 1234.777,A 0.000,B 0.000,C 90.000,E1 355.927} C_DIS
LIN {X 0.201,Y -526.683,Z 1234.773,A 0.000,B 0.000,C 90.000,E1 355.184} C_DIS
LIN {X 0.168,Y -529.692,Z 1234.770,A 0.000,B 0.000,C 90.000,E1 354.609} C_DIS
LIN {X -0.066,Y -533.098,Z 1234.766,A 0.000,B 0.000,C 90.000,E1 353.913} C_DIS
LIN {X -0.050,Y -535.644,Z 1234.763,A 0.000,B 0.000,C 90.000,E1 353.337} C_DIS
LIN {X -0.019,Y -538.016,Z 1234.760,A 0.000,B 0.000,C 90.000,E1 352.761} C_DIS
LIN {X 0.092,Y -541.222,Z 1234.755,A 0.000,B 0.000,C 90.000,E1 351.894} C_DIS
LIN {X 0.235,Y -544.214,Z 1234.750,A 0.000,B 0.000,C 90.000,E1 351.027} C_DIS
LIN {X -0.039,Y -546.896,Z 1234.746,A 0.000,B 0.000,C 90.000,E1 350.208} C_DIS
LIN {X -0.276,Y -550.089,Z 1234.739,A 0.000,B 0.000,C 90.000,E1 349.106} C_DIS
LIN {X 0.058,Y -552.316,Z 1234.735,A 0.000,B 0.000,C 90.000,E1 348.229} C_DIS
LIN {X -0.003,Y -554.991,Z 1234.729,A 0.000,B 0.000,C 90.000,E1 347.117} C_DIS
LIN {X 0.235,Y -557.984,Z 1234.721,A 0.000,B 0.000,C 90.000,E1 345.700} C_DIS
LIN {X -0.015,Y -560.596,Z 1234.713,A 0.000,B 0.000,C 90.000,E1 344.338} C_DIS
LIN {X 0.327,Y -562.485,Z 1234.707,A 0.000,B 0.000,C 90.000,E1 343.196} C_DIS
LIN {X -0.008,Y -564.060,Z 1234.701,A 0.000,B 0.000,C 90.000,E1 342.127} C_DIS
LIN {X 0.171,Y -565.730,Z 1234.693,A 0.000,B 0.000,C 90.000,E1 340.732} C_DIS
LIN {X 0.044,Y -566.604,Z 1234.687,A 0.000,B 0.000,C 90.000,E1 339.645} C_DIS
LIN {X -0.009,Y -567.005,Z 1234.682,A 0.000,B 0.000,C 90.000,E1 338.827} C_DIS
LIN {X 0.271,Y -567.133,Z 1234.678,A 0.000,B 0.000,C 90.000,E1 337.975} C_DIS
LIN {X 0.018,Y -566.927,Z 1234.673,A 0.000,B 0.000,C 90.000,E1 337.177} C_DIS
LIN {X -0.016,Y -566.369,Z 1234.669,A 0.000,B 0.000,C 90.000,E1 336.357} C_DIS
LIN {X 0.277,Y -565.095,Z 1234.663,A 0.000,B 0.000,C 90.000,E1 335.229} C_DIS
LIN {X -0.095,Y -564.218,Z 1234.660,A 0.000,B 0.000,C 90.000,E1 334.717} C_DIS
LIN {X -0.153,Y -562.691,Z 1234.655,A 0.000,B 0.000,C 90.000,E1 333.896} C_DIS
LIN {X -0.176,Y -560.095,Z 1234.649,A 0.000,B 0.000,C 90.000,E1 332.794} C_DIS
LIN {X -0.023,Y -557.615,Z 1234.644,A 0.000,B 0.000,C 90.000,E1 331.948} C_DIS
LIN {X 0.260,Y -556.711,Z 1234.643,A 0.000,B 0.000,C 90.000,E1 331.641} C_DIS
LIN {X -0.166,Y -554.614,Z 1234.640,A 0.000,B 0.000,C 90.000,E1 331.129} C_DIS
LIN {X 0.191,Y -550.893,Z 1234.635,A 0.000,B 0.000,C 90.000,E1 330.255} C_DIS
LIN {X -0.124,Y -547.393,Z 1234.631,A 0.000,B 0.000,C 90.000,E1 329.587} C_DIS
LIN {X 0.130,Y -544.154,Z 1234.628,A 0.000,B 0.000,C 90.000,E1 328.997} C_DIS
LIN {X -0.241,Y -539.642,Z 1234.624,A 0.000,B 0.000,C 90.000,E1 328.329} C_DIS
LIN {X 0.090,Y -534.758,Z 1234.620,A 0.000,B 0.000,C 90.000,E1 327.582} C_DIS
LIN {X 0.217,Y -528.493,Z 1234.615,A 0.000,B 0.000,C 90.000,E1 326.707} C_DIS
LIN {X 0.114,Y -515.731,Z 1234.606,A 0.000,B 0.000,C 90.000,E1 325.022} C_DIS
LIN {X -0.124,Y -512.510,Z 1234.603,A 0.000,B 0.000,C 90.000,E1 324.529} C_DIS
LIN {X -0.108,Y -510.072,Z 1234.600,A 0.000,B 0.000,C 90.000,E1 324.036} C_DIS
LIN {X 0.114,Y -509.453,Z 1234.599,A 0.000,B 0.000,C 90.000,E1 323.863} C_DIS
LIN {X -0.240,Y -507.387,Z 1234.595,A 0.000,B 0.000,C 90.000,E1 323.130} C_DIS
LIN {X 0.181,Y -506.208,Z 1234.590,A 0.000,B 0.000,C 90.000,E1 322.190} C_DIS
LIN {X -0.127,Y -505.705,Z 1234.585,A 0.000,B 0.000,C 90.000,E1 321.331} C_DIS
LIN {X 0.118,Y -507.065,Z 1234.569,A 0.000,B 0.000,C 90.000,E1 318.324} C_DIS
LIN {X -0.124,Y -507.664,Z 1234.560,A 0.000,B 0.000,C 90.000,E1 316.863} C_DIS
LIN {X -0.014,Y -508.193,Z 1234.552,A 0.000,B 0.000,C 90.000,E1 315.364} C_DIS
LIN {X 0.105,Y -508.723,Z 1234.544,A 0.000,B 0.000,C 90.000,E1 313.866} C_DIS
LIN {X 0.137,Y -509.376,Z 1234.534,A 0.000,B 0.000,C 90.000,E1 312.081} C_DIS
LIN {X 0.037,Y -509.862,Z 1234.527,A 0.000,B 0.000,C 90.000,E1 310.906} C_DIS
LIN {X 0.139,Y -510.492,Z 1234.517,A 0.000,B 0.000,C 90.000,E1 309.116} C_DIS
LIN {X 0.106,Y -510.827,Z 1234.511,A 0.000,B 0.000,C 90.000,E1 307.935} C_DIS
LIN {X 0.089,Y -511.287,Z 1234.503,A 0.000,B 0.000,C 90.000,E1 306.457} C_DIS
LIN {X 0.008,Y -511.726,Z 1234.493,A 0.000,B 0.000,C 90.000,E1 304.692} C_DIS
LIN {X 0.007,Y -512.089,Z 1234.485,A 0.000,B 0.000,C 90.000,E1 303.214} C_DIS
LIN {X -0.120,Y -512.264,Z 1234.476,A 0.000,B 0.000,C 90.000,E1 301.750} C_DIS
LIN {X 0.118,Y -512.415,Z 1234.467,A 0.000,B 0.000,C 90.000,E1 299.951} C_DIS
LIN {X 0.004,Y -512.478,Z 1234.458,A 0.000,B 0.000,C 90.000,E1 298.487} C_DIS
LIN {X -0.260,Y -512.489,Z 1234.448,A 0.000,B 0.000,C 90.000,E1 296.744} C_DIS
LIN {X 0.159,Y -512.577,Z 1234.435,A 0.000,B 0.000,C 90.000,E1 294.335} C_DIS
LIN {X 0.161,Y -512.697,Z 1234.429,A 0.000,B 0.000,C 90.000,E1 293.153} C_DIS
LIN {X 0.166,Y -512.437,Z 1234.422,A 0.000,B 0.000,C 90.000,E1 291.972} C_DIS
LIN {X 0.161,Y -512.034,Z 1234.416,A 0.000,B 0.000,C 90.000,E1 290.791} C_DIS
LIN {X 0.018,Y -511.231,Z 1234.406,A 0.000,B 0.000,C 90.000,E1 289.033} C_DIS
LIN {X -0.245,Y -510.675,Z 1234.398,A 0.000,B 0.000,C 90.000,E1 287.583} C_DIS
LIN {X -0.037,Y -509.597,Z 1234.384,A 0.000,B 0.000,C 90.000,E1 285.190} C_DIS
LIN {X -0.004,Y -508.739,Z 1234.376,A 0.000,B 0.000,C 90.000,E1 283.703} C_DIS
LIN {X -0.136,Y -508.129,Z 1234.371,A 0.000,B 0.000,C 90.000,E1 282.827} C_DIS
LIN {X 0.182,Y -507.339,Z 1234.365,A 0.000,B 0.000,C 90.000,E1 281.602} C_DIS
LIN {X 0.047,Y -505.003,Z 1234.346,A 0.000,B 0.000,C 90.000,E1 278.341} C_DIS
LIN {X 0.049,Y -503.860,Z 1234.336,A 0.000,B 0.000,C 90.000,E1 276.549} C_DIS
LIN {X 0.092,Y -503.102,Z 1234.328,A 0.000,B 0.000,C 90.000,E1 275.049} C_DIS
LIN {X -0.049,Y -502.090,Z 1234.318,A 0.000,B 0.000,C 90.000,E1 273.269} C_DIS
LIN {X -0.098,Y -501.075,Z 1234.310,A 0.000,B 0.000,C 90.000,E1 271.776} C_DIS
LIN {X -0.081,Y -500.089,Z 1234.303,A 0.000,B 0.000,C 90.000,E1 270.573} C_DIS
LIN {X -0.199,Y -499.171,Z 1234.295,A 0.000,B 0.000,C 90.000,E1 269.083} C_DIS
LIN {X -0.067,Y -498.529,Z 1234.290,A 0.000,B 0.000,C 90.000,E1 268.165} C_DIS
LIN {X 0.165,Y -497.580,Z 1234.280,A 0.000,B 0.000,C 90.000,E1 266.331} C_DIS
LIN {X -0.060,Y -496.498,Z 1234.270,A 0.000,B 0.000,C 90.000,E1 264.546} C_DIS
LIN {X -0.055,Y -495.586,Z 1234.263,A 0.000,B 0.000,C 90.000,E1 263.337} C_DIS
LIN {X 0.088,Y -494.867,Z 1234.258,A 0.000,B 0.000,C 90.000,E1 262.413} C_DIS
LIN {X 0.029,Y -493.475,Z 1234.250,A 0.000,B 0.000,C 90.000,E1 260.905} C_DIS
LIN {X 0.218,Y -491.469,Z 1234.238,A 0.000,B 0.000,C 90.000,E1 258.757} C_DIS
LIN {X 0.058,Y -489.847,Z 1234.226,A 0.000,B 0.000,C 90.000,E1 256.645} C_DIS
LIN {X -0.030,Y -488.535,Z 1234.214,A 0.000,B 0.000,C 90.000,E1 254.519} C_DIS
LIN {X 0.124,Y -487.093,Z 1234.200,A 0.000,B 0.000,C 90.000,E1 252.054} C_DIS
LIN {X -0.093,Y -486.193,Z 1234.190,A 0.000,B 0.000,C 90.000,E1 250.242} C_DIS
LIN {X -0.200,Y -485.581,Z 1234.183,A 0.000,B 0.000,C 90.000,E1 249.028} C_DIS
LIN {X -0.136,Y -484.738,Z 1234.175,A 0.000,B 0.000,C 90.000,E1 247.486} C_DIS
LIN {X 0.101,Y -483.699,Z 1234.166,A 0.000,B 0.000,C 90.000,E1 245.921} C_DIS
LIN {X 0.083,Y -482.270,Z 1234.156,A 0.000,B 0.000,C 90.000,E1 244.076} C_DIS
LIN {X 0.046,Y -481.103,Z 1234.147,A 0.000,B 0.000,C 90.000,E1 242.538} C_DIS
LIN {X 0.181,Y -479.432,Z 1234.137,A 0.000,B 0.000,C 90.000,E1 240.667} C_DIS
LIN {X 0.126,Y -477.858,Z 1234.129,A 0.000,B 0.000,C 90.000,E1 239.125} C_DIS
LIN {X 0.047,Y -476.226,Z 1234.120,A 0.000,B 0.000,C 90.000,E1 237.582} C_DIS
LIN {X 0.192,Y -474.708,Z 1234.111,A 0.000,B 0.000,C 90.000,E1 236.008} C_DIS
LIN {X 0.141,Y -472.547,Z 1234.099,A 0.000,B 0.000,C 90.000,E1 233.829} C_DIS
LIN {X -0.130,Y -471.677,Z 1234.094,A 0.000,B 0.000,C 90.000,E1 232.924} C_DIS
LIN {X 0.153,Y -469.921,Z 1234.083,A 0.000,B 0.000,C 90.000,E1 231.009} C_DIS
LIN {X -0.032,Y -468.566,Z 1234.075,A 0.000,B 0.000,C 90.000,E1 229.461} C_DIS
LIN {X 0.122,Y -467.035,Z 1234.064,A 0.000,B 0.000,C 90.000,E1 227.553} C_DIS
LIN {X 0.215,Y -465.608,Z 1234.054,A 0.000,B 0.000,C 90.000,E1 225.648} C_DIS
LIN {X 0.122,Y -463.851,Z 1234.029,A 0.000,B 0.000,C 90.000,E1 221.229} C_DIS
LIN {X -0.044,Y -465.418,Z 1233.996,A 0.000,B 0.000,C 90.000,E1 215.231} C_DIS
LIN {X 0.205,Y -466.929,Z 1233.982,A 0.000,B 0.000,C 90.000,E1 212.673} C_DIS
LIN {X 0.085,Y -468.744,Z 1233.971,A 0.000,B 0.000,C 90.000,E1 210.797} C_DIS
LIN {X 0.043,Y -471.781,Z 1233.955,A 0.000,B 0.000,C 90.000,E1 207.975} C_DIS
LIN {X 0.123,Y -474.892,Z 1233.942,A 0.000,B 0.000,C 90.000,E1 205.463} C_DIS
LIN {X -0.154,Y -479.438,Z 1233.924,A 0.000,B 0.000,C 90.000,E1 202.386} C_DIS
LIN {X 0.258,Y -481.486,Z 1233.917,A 0.000,B 0.000,C 90.000,E1 201.099} C_DIS
LIN {X -0.162,Y -488.071,Z 1233.899,A 0.000,B 0.000,C 90.000,E1 197.764} C_DIS
LIN {X 0.041,Y -493.645,Z 1233.885,A 0.000,B 0.000,C 90.000,E1 195.300} C_DIS
LIN {X 0.156,Y -497.364,Z 1233.877,A 0.000,B 0.000,C 90.000,E1 193.772} C_DIS
LIN {X -0.210,Y -502.011,Z 1233.867,A 0.000,B 0.000,C 90.000,E1 192.007} C_DIS
LIN {X 0.217,Y -510.025,Z 1233.850,A 0.000,B 0.000,C 90.000,E1 188.973} C_DIS
LIN {X -0.120,Y -514.178,Z 1233.842,A 0.000,B 0.000,C 90.000,E1 187.530} C_DIS
LIN {X 0.116,Y -518.949,Z 1233.832,A 0.000,B 0.000,C 90.000,E1 185.739} C_DIS
LIN {X -0.053,Y -522.206,Z 1233.826,A 0.000,B 0.000,C 90.000,E1 184.588} C_DIS
LIN {X 0.260,Y -526.999,Z 1233.816,A 0.000,B 0.000,C 90.000,E1 182.808} C_DIS
LIN {X 0.145,Y -530.984,Z 1233.808,A 0.000,B 0.000,C 90.000,E1 181.375} C_DIS
LIN {X 0.091,Y -534.847,Z 1233.800,A 0.000,B 0.000,C 90.000,E1 179.943} C_DIS
LIN {X 0.106,Y -538.657,Z 1233.792,A 0.000,B 0.000,C 90.000,E1 178.511} C_DIS
LIN {X 0.201,Y -542.280,Z 1233.784,A 0.000,B 0.000,C 90.000,E1 177.078} C_DIS
LIN {X -0.241,Y -544.403,Z 1233.779,A 0.000,B 0.000,C 90.000,E1 176.274} C_DIS
LIN {X 0.076,Y -548.447,Z 1233.770,A 0.000,B 0.000,C 90.000,E1 174.546} C_DIS
LIN {X -0.166,Y -551.652,Z 1233.762,A 0.000,B 0.000,C 90.000,E1 173.166} C_DIS
LIN {X -0.174,Y -555.376,Z 1233.753,A 0.000,B 0.000,C 90.000,E1 171.489} C_DIS
LIN {X -0.155,Y -558.411,Z 1233.745,A 0.000,B 0.000,C 90.000,E1 170.095} C_DIS
LIN {X -0.235,Y -560.792,Z 1233.739,A 0.000,B 0.000,C 90.000,E1 168.993} C_DIS
LIN {X -0.252,Y -564.919,Z 1233.728,A 0.000,B 0.000,C 90.000,E1 167.061} C_DIS
LIN {X 0.104,Y -569.125,Z 1233.717,A 0.000,B 0.000,C 90.000,E1 165.102} C_DIS
LIN {X 0.238,Y -578.974,Z 1233.696,A 0.000,B 0.000,C 90.000,E1 161.275} C_DIS
LIN {X 0.214,Y -585.317,Z 1233.686,A 0.000,B 0.000,C 90.000,E1 159.390} C_DIS
LIN {X -0.076,Y -597.259,Z 1233.669,A 0.000,B 0.000,C 90.000,E1 156.485} C_DIS
LIN {X 0.073,Y -602.806,Z 1233.662,A 0.000,B 0.000,C 90.000,E1 155.153} C_DIS
LIN {X 0.060,Y -608.407,Z 1233.655,A 0.000,B 0.000,C 90.000,E1 153.845} C_DIS
LIN {X 0.162,Y -612.630,Z 1233.649,A 0.000,B 0.000,C 90.000,E1 152.794} C_DIS
LIN {X 0.099,Y -614.704,Z 1233.646,A 0.000,B 0.000,C 90.000,E1 152.281} C_DIS
LIN {X -0.010,Y -619.670,Z 1233.639,A 0.000,B 0.000,C 90.000,E1 151.001} C_DIS
LIN {X 0.029,Y -625.418,Z 1233.630,A 0.000,B 0.000,C 90.000,E1 149.459} C_DIS
LIN {X 0.367,Y -628.350,Z 1233.626,A 0.000,B 0.000,C 90.000,E1 148.663} C_DIS
LIN {X -0.303,Y -632.954,Z 1233.619,A 0.000,B 0.000,C 90.000,E1 147.454} C_DIS
LIN {X -0.032,Y -637.305,Z 1233.612,A 0.000,B 0.000,C 90.000,E1 146.167} C_DIS
LIN {X 0.140,Y -641.415,Z 1233.605,A 0.000,B 0.000,C 90.000,E1 144.895} C_DIS
LIN {X 0.086,Y -643.650,Z 1233.601,A 0.000,B 0.000,C 90.000,E1 144.149} C_DIS
LIN {X 0.327,Y -646.461,Z 1233.595,A 0.000,B 0.000,C 90.000,E1 143.130} C_DIS
LIN {X 0.138,Y -649.670,Z 1233.589,A 0.000,B 0.000,C 90.000,E1 141.904} C_DIS
LIN {X -0.066,Y -653.303,Z 1233.580,A 0.000,B 0.000,C 90.000,E1 140.436} C_DIS
LIN {X -0.239,Y -656.178,Z 1233.573,A 0.000,B 0.000,C 90.000,E1 139.218} C_DIS
LIN {X 0.098,Y -659.585,Z 1233.565,A 0.000,B 0.000,C 90.000,E1 137.715} C_DIS
LIN {X -0.032,Y -664.091,Z 1233.554,A 0.000,B 0.000,C 90.000,E1 135.769} C_DIS
LIN {X 0.414,Y -668.934,Z 1233.543,A 0.000,B 0.000,C 90.000,E1 133.785} C_DIS
LIN {X 0.015,Y -672.665,Z 1233.535,A 0.000,B 0.000,C 90.000,E1 132.366} C_DIS
LIN {X 0.180,Y -676.362,Z 1233.527,A 0.000,B 0.000,C 90.000,E1 130.906} C_DIS
LIN {X -0.054,Y -679.450,Z 1233.521,A 0.000,B 0.000,C 90.000,E1 129.725} C_DIS
LIN {X 0.365,Y -683.712,Z 1233.511,A 0.000,B 0.000,C 90.000,E1 128.016} C_DIS
LIN {X 0.412,Y -687.352,Z 1233.504,A 0.000,B 0.000,C 90.000,E1 126.583} C_DIS
LIN {X -0.109,Y -689.616,Z 1233.498,A 0.000,B 0.000,C 90.000,E1 125.678} C_DIS
LIN {X 0.008,Y -692.297,Z 1233.492,A 0.000,B 0.000,C 90.000,E1 124.485} C_DIS
LIN {X -0.190,Y -695.457,Z 1233.484,A 0.000,B 0.000,C 90.000,E1 123.086} C_DIS
LIN {X -0.035,Y -697.376,Z 1233.479,A 0.000,B 0.000,C 90.000,E1 122.133} C_DIS
LIN {X 0.398,Y -699.667,Z 1233.472,A 0.000,B 0.000,C 90.000,E1 120.924} C_DIS
LIN {X -0.092,Y -701.819,Z 1233.466,A 0.000,B 0.000,C 90.000,E1 119.795} C_DIS
LIN {X 0.118,Y -703.040,Z 1233.462,A 0.000,B 0.000,C 90.000,E1 119.077} C_DIS
LIN {X 0.341,Y -704.076,Z 1233.458,A 0.000,B 0.000,C 90.000,E1 118.359} C_DIS
LIN {X -0.090,Y -705.156,Z 1233.453,A 0.000,B 0.000,C 90.000,E1 117.462} C_DIS
LIN {X -0.187,Y -705.804,Z 1233.447,A 0.000,B 0.000,C 90.000,E1 116.539} C_DIS
LIN {X -0.258,Y -706.073,Z 1233.443,A 0.000,B 0.000,C 90.000,E1 115.848} C_DIS
LIN {X -0.322,Y -706.051,Z 1233.440,A 0.000,B 0.000,C 90.000,E1 115.155} C_DIS
LIN {X 0.262,Y -705.697,Z 1233.437,A 0.000,B 0.000,C 90.000,E1 114.643} C_DIS
LIN {X -0.094,Y -704.997,Z 1233.434,A 0.000,B 0.000,C 90.000,E1 114.207} C_DIS
LIN {X 0.195,Y -704.587,Z 1233.433,A 0.000,B 0.000,C 90.000,E1 113.951} C_DIS
LIN {X -0.166,Y -702.503,Z 1233.431,A 0.000,B 0.000,C 90.000,E1 113.515} C_DIS
LIN {X 0.112,Y -701.273,Z 1233.429,A 0.000,B 0.000,C 90.000,E1 113.259} C_DIS
LIN {X -0.026,Y -700.244,Z 1233.429,A 0.000,B 0.000,C 90.000,E1 113.153} C_DIS
LIN {X 0.012,Y -695.300,Z 1233.426,A 0.000,B 0.000,C 90.000,E1 112.695} C_DIS
LIN {X -0.079,Y -693.406,Z 1233.426,A 0.000,B 0.000,C 90.000,E1 112.589} C_DIS
LIN {X 0.176,Y -686.373,Z 1233.424,A 0.000,B 0.000,C 90.000,E1 112.333} C_DIS
LIN {X -0.158,Y -684.999,Z 1233.424,A 0.000,B 0.000,C 90.000,E1 112.333} C_DIS
LIN {X -0.135,Y -677.285,Z 1233.424,A 0.000,B 0.000,C 90.000,E1 112.280} C_DIS
LIN {X -0.186,Y -618.633,Z 1233.424,A 0.000,B 0.000,C 90.000,E1 112.280} C_DIS
LIN {X -0.091,Y -615.309,Z 1233.423,A 0.000,B 0.000,C 90.000,E1 112.078} C_DIS
LIN {X -0.361,Y -612.710,Z 1233.421,A 0.000,B 0.000,C 90.000,E1 111.844} C_DIS
LIN {X 0.165,Y -612.667,Z 1233.421,A 0.000,B 0.000,C 90.000,E1 111.791} C_DIS
LIN {X 0.066,Y -612.279,Z 1233.420,A 0.000,B 0.000,C 90.000,E1 111.663} C_DIS
LIN {X 0.228,Y -613.231,Z 1233.418,A 0.000,B 0.000,C 90.000,E1 111.227} C_DIS
LIN {X 0.185,Y -614.244,Z 1233.417,A 0.000,B 0.000,C 90.000,E1 110.972} C_DIS
LIN {X 0.240,Y -619.056,Z 1233.411,A 0.000,B 0.000,C 90.000,E1 109.939} C_DIS
LIN {X -0.262,Y -622.336,Z 1233.407,A 0.000,B 0.000,C 90.000,E1 109.214} C_DIS
LIN {X 0.005,Y -629.726,Z 1233.397,A 0.000,B 0.000,C 90.000,E1 107.402} C_DIS
LIN {X 0.018,Y -634.184,Z 1233.391,A 0.000,B 0.000,C 90.000,E1 106.386} C_DIS
LIN {X 0.091,Y -638.298,Z 1233.385,A 0.000,B 0.000,C 90.000,E1 105.371} C_DIS
LIN {X -0.246,Y -640.001,Z 1233.383,A 0.000,B 0.000,C 90.000,E1 104.898} C_DIS
LIN {X 0.211,Y -641.516,Z 1233.380,A 0.000,B 0.000,C 90.000,E1 104.356} C_DIS
LIN {X -0.107,Y -642.823,Z 1233.377,A 0.000,B 0.000,C 90.000,E1 103.883} C_DIS
LIN {X 0.059,Y -644.343,Z 1233.373,A 0.000,B 0.000,C 90.000,E1 103.119} C_DIS
LIN {X -0.241,Y -645.046,Z 1233.370,A 0.000,B 0.000,C 90.000,E1 102.647} C_DIS
LIN {X 0.092,Y -645.259,Z 1233.367,A 0.000,B 0.000,C 90.000,E1 102.119} C_DIS
LIN {X -0.335,Y -645.161,Z 1233.365,A 0.000,B 0.000,C 90.000,E1 101.658} C_DIS
LIN {X 0.151,Y -645.010,Z 1233.363,A 0.000,B 0.000,C 90.000,E1 101.366} C_DIS
LIN {X -0.146,Y -644.453,Z 1233.360,A 0.000,B 0.000,C 90.000,E1 100.894} C_DIS
LIN {X 0.182,Y -643.399,Z 1233.358,A 0.000,B 0.000,C 90.000,E1 100.366} C_DIS
LIN {X -0.243,Y -642.012,Z 1233.355,A 0.000,B 0.000,C 90.000,E1 99.905} C_DIS
LIN {X 0.065,Y -640.298,Z 1233.352,A 0.000,B 0.000,C 90.000,E1 99.378} C_DIS
LIN {X -0.204,Y -639.357,Z 1233.351,A 0.000,B 0.000,C 90.000,E1 99.151} C_DIS
LIN {X -0.055,Y -636.528,Z 1233.347,A 0.000,B 0.000,C 90.000,E1 98.511} C_DIS
LIN {X 0.254,Y -634.671,Z 1233.345,A 0.000,B 0.000,C 90.000,E1 98.106} C_DIS
LIN {X 0.063,Y -633.102,Z 1233.344,A 0.000,B 0.000,C 90.000,E1 97.871} C_DIS
LIN {X 0.062,Y -628.912,Z 1233.340,A 0.000,B 0.000,C 90.000,E1 97.239} C_DIS
LIN {X -0.294,Y -626.147,Z 1233.338,A 0.000,B 0.000,C 90.000,E1 96.891} C_DIS
LIN {X -0.194,Y -621.690,Z 1233.335,A 0.000,B 0.000,C 90.000,E1 96.372} C_DIS
LIN {X 0.034,Y -618.095,Z 1233.333,A 0.000,B 0.000,C 90.000,E1 95.967} C_DIS
LIN {X 0.209,Y -611.486,Z 1233.330,A 0.000,B 0.000,C 90.000,E1 95.334} C_DIS
LIN {X 0.298,Y -604.120,Z 1233.327,A 0.000,B 0.000,C 90.000,E1 94.759} C_DIS
LIN {X 0.226,Y -596.527,Z 1233.324,A 0.000,B 0.000,C 90.000,E1 94.245} C_DIS
LIN {X -0.024,Y -588.360,Z 1233.321,A 0.000,B 0.000,C 90.000,E1 93.784} C_DIS
LIN {X 0.077,Y -583.331,Z 1233.320,A 0.000,B 0.000,C 90.000,E1 93.498} C_DIS
LIN {X 0.203,Y -576.274,Z 1233.318,A 0.000,B 0.000,C 90.000,E1 93.154} C_DIS
LIN {X -0.274,Y -570.826,Z 1233.316,A 0.000,B 0.000,C 90.000,E1 92.980} C_DIS
LIN {X 0.054,Y -567.371,Z 1233.315,A 0.000,B 0.000,C 90.000,E1 92.751} C_DIS
LIN {X -0.002,Y -567.342,Z 1233.315,A 0.000,B 0.000,C 90.000,E1 92.751} C_DIS
LIN {X -0.114,Y -566.322,Z 1233.314,A 0.000,B 0.000,C 90.000,E1 92.465} C_DIS
LIN {X 0.270,Y -565.693,Z 1233.313,A 0.000,B 0.000,C 90.000,E1 92.293} C_DIS
LIN {X 0.229,Y -565.679,Z 1233.313,A 0.000,B 0.000,C 90.000,E1 92.293} C_DIS
LIN {X 0.249,Y -565.523,Z 1233.310,A 0.000,B 0.000,C 90.000,E1 91.776} C_DIS
LIN {X -0.073,Y -567.200,Z 1233.296,A 0.000,B 0.000,C 90.000,E1 89.198} C_DIS
LIN {X -0.025,Y -568.174,Z 1233.288,A 0.000,B 0.000,C 90.000,E1 87.822} C_DIS
LIN {X -0.245,Y -569.738,Z 1233.277,A 0.000,B 0.000,C 90.000,E1 85.927} C_DIS
LIN {X -0.262,Y -571.706,Z 1233.265,A 0.000,B 0.000,C 90.000,E1 83.742} C_DIS
LIN {X 0.156,Y -573.317,Z 1233.256,A 0.000,B 0.000,C 90.000,E1 82.064} C_DIS
LIN {X -0.160,Y -574.560,Z 1233.249,A 0.000,B 0.000,C 90.000,E1 80.735} C_DIS
LIN {X -0.011,Y -575.421,Z 1233.242,A 0.000,B 0.000,C 90.000,E1 79.634} C_DIS
LIN {X -0.241,Y -576.721,Z 1233.232,A 0.000,B 0.000,C 90.000,E1 77.757} C_DIS
LIN {X 0.258,Y -577.570,Z 1233.224,A 0.000,B 0.000,C 90.000,E1 76.353} C_DIS
LIN {X -0.004,Y -578.523,Z 1233.215,A 0.000,B 0.000,C 90.000,E1 74.755} C_DIS
LIN {X -0.091,Y -579.399,Z 1233.206,A 0.000,B 0.000,C 90.000,E1 73.142} C_DIS
LIN {X -0.021,Y -580.015,Z 1233.200,A 0.000,B 0.000,C 90.000,E1 72.054} C_DIS
LIN {X 0.105,Y -581.062,Z 1233.191,A 0.000,B 0.000,C 90.000,E1 70.423} C_DIS
LIN {X -0.287,Y -583.169,Z 1233.173,A 0.000,B 0.000,C 90.000,E1 67.230} C_DIS
LIN {X 0.171,Y -584.811,Z 1233.163,A 0.000,B 0.000,C 90.000,E1 65.305} C_DIS
LIN {X -0.014,Y -586.738,Z 1233.151,A 0.000,B 0.000,C 90.000,E1 63.179} C_DIS
LIN {X -0.018,Y -588.607,Z 1233.141,A 0.000,B 0.000,C 90.000,E1 61.307} C_DIS
LIN {X -0.290,Y -589.995,Z 1233.133,A 0.000,B 0.000,C 90.000,E1 59.999} C_DIS
LIN {X -0.243,Y -591.380,Z 1233.126,A 0.000,B 0.000,C 90.000,E1 58.663} C_DIS
LIN {X 0.030,Y -592.845,Z 1233.117,A 0.000,B 0.000,C 90.000,E1 57.041} C_DIS
LIN {X -0.270,Y -593.827,Z 1233.111,A 0.000,B 0.000,C 90.000,E1 56.008} C_DIS
LIN {X -0.337,Y -594.921,Z 1233.104,A 0.000,B 0.000,C 90.000,E1 54.689} C_DIS
LIN {X -0.041,Y -595.965,Z 1233.096,A 0.000,B 0.000,C 90.000,E1 53.336} C_DIS
LIN {X 0.266,Y -597.430,Z 1233.086,A 0.000,B 0.000,C 90.000,E1 51.457} C_DIS
LIN {X 0.121,Y -597.965,Z 1233.082,A 0.000,B 0.000,C 90.000,E1 50.678} C_DIS
LIN {X 0.144,Y -598.969,Z 1233.070,A 0.000,B 0.000,C 90.000,E1 48.566} C_DIS
LIN {X -0.281,Y -599.420,Z 1233.064,A 0.000,B 0.000,C 90.000,E1 47.553} C_DIS
LIN {X -0.063,Y -599.678,Z 1233.057,A 0.000,B 0.000,C 90.000,E1 46.215} C_DIS
LIN {X -0.060,Y -599.752,Z 1233.051,A 0.000,B 0.000,C 90.000,E1 45.162} C_DIS
LIN {X -0.045,Y -599.535,Z 1233.042,A 0.000,B 0.000,C 90.000,E1 43.581} C_DIS
LIN {X 0.166,Y -599.304,Z 1233.038,A 0.000,B 0.000,C 90.000,E1 42.771} C_DIS
LIN {X -0.021,Y -598.666,Z 1233.030,A 0.000,B 0.000,C 90.000,E1 41.472} C_DIS
LIN {X 0.014,Y -597.844,Z 1233.022,A 0.000,B 0.000,C 90.000,E1 39.886} C_DIS
LIN {X 0.021,Y -597.584,Z 1233.019,A 0.000,B 0.000,C 90.000,E1 39.358} C_DIS
LIN {X 0.256,Y -596.997,Z 1233.014,A 0.000,B 0.000,C 90.000,E1 38.543} C_DIS
LIN {X -0.354,Y -596.195,Z 1233.010,A 0.000,B 0.000,C 90.000,E1 37.810} C_DIS
LIN {X -0.043,Y -594.683,Z 1233.003,A 0.000,B 0.000,C 90.000,E1 36.457} C_DIS
LIN {X 0.147,Y -593.570,Z 1232.998,A 0.000,B 0.000,C 90.000,E1 35.644} C_DIS
LIN {X -0.154,Y -591.826,Z 1232.992,A 0.000,B 0.000,C 90.000,E1 34.612} C_DIS
LIN {X 0.347,Y -589.687,Z 1232.986,A 0.000,B 0.000,C 90.000,E1 33.499} C_DIS
LIN {X -0.196,Y -587.838,Z 1232.982,A 0.000,B 0.000,C 90.000,E1 32.752} C_DIS
LIN {X 0.053,Y -585.604,Z 1232.977,A 0.000,B 0.000,C 90.000,E1 31.926} C_DIS
LIN {X -0.164,Y -582.104,Z 1232.971,A 0.000,B 0.000,C 90.000,E1 30.875} C_DIS
LIN {X 0.013,Y -578.974,Z 1232.967,A 0.000,B 0.000,C 90.000,E1 30.050} C_DIS
LIN {X -0.348,Y -575.997,Z 1232.963,A 0.000,B 0.000,C 90.000,E1 29.411} C_DIS
LIN {X -0.028,Y -572.083,Z 1232.959,A 0.000,B 0.000,C 90.000,E1 28.565} C_DIS
LIN {X 0.157,Y -566.868,Z 1232.953,A 0.000,B 0.000,C 90.000,E1 27.590} C_DIS
LIN {X -0.111,Y -564.472,Z 1232.951,A 0.000,B 0.000,C 90.000,E1 27.206} C_DIS
LIN {X 0.271,Y -561.061,Z 1232.948,A 0.000,B 0.000,C 90.000,E1 26.616} C_DIS
LIN {X 0.062,Y -554.616,Z 1232.943,A 0.000,B 0.000,C 90.000,E1 25.668} C_DIS
LIN {X 0.124,Y -550.598,Z 1232.940,A 0.000,B 0.000,C 90.000,E1 25.103} C_DIS
LIN {X 0.141,Y -543.864,Z 1232.935,A 0.000,B 0.000,C 90.000,E1 24.259} C_DIS
LIN {X -0.145,Y -536.627,Z 1232.930,A 0.000,B 0.000,C 90.000,E1 23.439} C_DIS
LIN {X 0.276,Y -531.582,Z 1232.927,A 0.000,B 0.000,C 90.000,E1 22.823} C_DIS
LIN {X -0.130,Y -523.750,Z 1232.922,A 0.000,B 0.000,C 90.000,E1 22.025} C_DIS
LIN {X -0.082,Y -518.465,Z 1232.919,A 0.000,B 0.000,C 90.000,E1 21.461} C_DIS
LIN {X -0.036,Y -507.761,Z 1232.913,A 0.000,B 0.000,C 90.000,E1 20.375} C_DIS
LIN {X 0.202,Y -497.851,Z 1232.908,A 0.000,B 0.000,C 90.000,E1 19.396} C_DIS
LIN {X 0.193,Y -490.711,Z 1232.904,A 0.000,B 0.000,C 90.000,E1 18.725} C_DIS
LIN {X 0.024,Y -478.946,Z 1232.898,A 0.000,B 0.000,C 90.000,E1 17.692} C_DIS
LIN {X -0.176,Y -467.224,Z 1232.893,A 0.000,B 0.000,C 90.000,E1 16.677} C_DIS
LIN {X -0.050,Y -450.863,Z 1232.884,A 0.000,B 0.000,C 90.000,E1 15.190} C_DIS
LIN {X -0.177,Y -436.367,Z 1232.877,A 0.000,B 0.000,C 90.000,E1 13.828} C_DIS
LIN {X 0.142,Y -416.406,Z 1232.865,A 0.000,B 0.000,C 90.000,E1 11.715} C_DIS
LIN {X 0.140,Y -399.751,Z 1232.855,A 0.000,B 0.000,C 90.000,E1 9.792} C_DIS
LIN {X 0.168,Y -395.897,Z 1232.851,A 0.000,B 0.000,C 90.000,E1 9.208} C_DIS
LIN {X 0.050,Y -394.087,Z 1232.849,A 0.000,B 0.000,C 90.000,E1 8.803} C_DIS
LIN {X 0.013,Y -394.071,Z 1232.849,A 0.000,B 0.000,C 90.000,E1 8.803} C_DIS
LIN {X -0.136,Y -394.027,Z 1232.848,A 0.000,B 0.000,C 90.000,E1 8.681} C_DIS
LIN {X 0.216,Y -394.041,Z 1232.848,A 0.000,B 0.000,C 90.000,E1 8.624} C_DIS
LIN {X -0.172,Y -396.699,Z 1232.845,A 0.000,B 0.000,C 90.000,E1 8.106} C_DIS
LIN {X 0.074,Y -400.498,Z 1232.843,A 0.000,B 0.000,C 90.000,E1 7.644} C_DIS
LIN {X 0.145,Y -406.083,Z 1232.840,A 0.000,B 0.000,C 90.000,E1 7.182} C_DIS
LIN {X -0.211,Y -413.865,Z 1232.837,A 0.000,B 0.000,C 90.000,E1 6.663} C_DIS
LIN {X -0.001,Y -420.553,Z 1232.834,A 0.000,B 0.000,C 90.000,E1 6.144} C_DIS
LIN {X 0.045,Y -423.831,Z 1232.833,A 0.000,B 0.000,C 90.000,E1 5.910} C_DIS
LIN {X -0.155,Y -433.135,Z 1232.829,A 0.000,B 0.000,C 90.000,E1 5.220} C_DIS
LIN {X 0.136,Y -447.414,Z 1232.823,A 0.000,B 0.000,C 90.000,E1 4.073} C_DIS
LIN {X -0.197,Y -456.800,Z 1232.819,A 0.000,B 0.000,C 90.000,E1 3.383} C_DIS
LIN {X -0.151,Y -466.070,Z 1232.815,A 0.000,B 0.000,C 90.000,E1 2.636} C_DIS
LIN {X -0.078,Y -472.110,Z 1232.812,A 0.000,B 0.000,C 90.000,E1 2.121} C_DIS
LIN {X 0.146,Y -479.347,Z 1232.808,A 0.000,B 0.000,C 90.000,E1 1.432} C_DIS
LIN {X -0.146,Y -485.025,Z 1232.805,A 0.000,B 0.000,C 90.000,E1 0.917} C_DIS
LIN {X 0.128,Y -492.721,Z 1232.800,A 0.000,B 0.000,C 90.000,E1 0.057} C_DIS
LIN {X 0.104,Y -497.801,Z 1232.797,A 0.000,B 0.000,C 90.000,E1 359.484} C_DIS
LIN {X 0.139,Y -503.745,Z 1232.793,A 0.000,B 0.000,C 90.000,E1 358.740} C_DIS
LIN {X 0.233,Y -509.279,Z 1232.789,A 0.000,B 0.000,C 90.000,E1 357.993} C_DIS
LIN {X -0.249,Y -514.444,Z 1232.785,A 0.000,B 0.000,C 90.000,E1 357.306} C_DIS
LIN {X -0.152,Y -519.212,Z 1232.781,A 0.000,B 0.000,C 90.000,E1 356.560} C_DIS
LIN {X -0.276,Y -522.799,Z 1232.778,A 0.000,B 0.000,C 90.000,E1 355.988} C_DIS
LIN {X -0.101,Y -526.881,Z 1232.774,A 0.000,B 0.000,C 90.000,E1 355.241} C_DIS
LIN {X -0.134,Y -529.901,Z 1232.770,A 0.000,B 0.000,C 90.000,E1 354.666} C_DIS
LIN {X 0.163,Y -533.347,Z 1232.766,A 0.000,B 0.000,C 90.000,E1 353.913} C_DIS
LIN {X 0.183,Y -535.900,Z 1232.763,A 0.000,B 0.000,C 90.000,E1 353.337} C_DIS
LIN {X 0.276,Y -539.393,Z 1232.758,A 0.000,B 0.000,C 90.000,E1 352.470} C_DIS
LIN {X -0.132,Y -542.549,Z 1232.754,A 0.000,B 0.000,C 90.000,E1 351.659} C_DIS
LIN {X 0.026,Y -545.442,Z 1232.749,A 0.000,B 0.000,C 90.000,E1 350.792} C_DIS
LIN {X 0.212,Y -548.011,Z 1232.744,A 0.000,B 0.000,C 90.000,E1 349.926} C_DIS
LIN {X 0.088,Y -551.139,Z 1232.738,A 0.000,B 0.000,C 90.000,E1 348.814} C_DIS
LIN {X 0.013,Y -553.990,Z 1232.732,A 0.000,B 0.000,C 90.000,E1 347.701} C_DIS
LIN {X -0.153,Y -555.929,Z 1232.727,A 0.000,B 0.000,C 90.000,E1 346.881} C_DIS
LIN {X 0.102,Y -558.872,Z 1232.719,A 0.000,B 0.000,C 90.000,E1 345.463} C_DIS
LIN {X -0.135,Y -561.462,Z 1232.712,A 0.000,B 0.000,C 90.000,E1 344.102} C_DIS
LIN {X 0.218,Y -563.273,Z 1232.706,A 0.000,B 0.000,C 90.000,E1 342.960} C_DIS
LIN {X 0.066,Y -564.838,Z 1232.699,A 0.000,B 0.000,C 90.000,E1 341.873} C_DIS
LIN {X -0.063,Y -566.186,Z 1232.693,A 0.000,B 0.000,C 90.000,E1 340.786} C_DIS
LIN {X -0.180,Y -567.123,Z 1232.687,A 0.000,B 0.000,C 90.000,E1 339.699} C_DIS
LIN {X 0.099,Y -567.580,Z 1232.683,A 0.000,B 0.000,C 90.000,E1 338.847} C_DIS
LIN {X 0.062,Y -567.747,Z 1232.678,A 0.000,B 0.000,C 90.000,E1 338.028} C_DIS
LIN {X -0.180,Y -567.594,Z 1232.673,A 0.000,B 0.000,C 90.000,E1 337.230} C_DIS
LIN {X 0.315,Y -567.087,Z 1232.669,A 0.000,B 0.000,C 90.000,E1 336.357} C_DIS
LIN {X 0.288,Y -566.254,Z 1232.664,A 0.000,B 0.000,C 90.000,E1 335.537} C_DIS
LIN {X -0.076,Y -565.530,Z 1232.661,A 0.000,B 0.000,C 90.000,E1 335.025} C_DIS
LIN {X -0.118,Y -564.093,Z 1232.657,A 0.000,B 0.000,C 90.000,E1 334.204} C_DIS
LIN {X 0.012,Y -563.032,Z 1232.654,A 0.000,B 0.000,C 90.000,E1 333.640} C_DIS
LIN {X -0.005,Y -560.294,Z 1232.647,A 0.000,B 0.000,C 90.000,E1 332.538} C_DIS
LIN {X 0.089,Y -558.751,Z 1232.644,A 0.000,B 0.000,C 90.000,E1 331.975} C_DIS
LIN {X -0.268,Y -555.715,Z 1232.640,A 0.000,B 0.000,C 90.000,E1 331.179} C_DIS
LIN {X -0.282,Y -551.413,Z 1232.634,A 0.000,B 0.000,C 90.000,E1 330.205} C_DIS
LIN {X 0.159,Y -547.910,Z 1232.630,A 0.000,B 0.000,C 90.000,E1 329.459} C_DIS
LIN {X -0.181,Y -543.714,Z 1232.627,A 0.000,B 0.000,C 90.000,E1 328.791} C_DIS
LIN {X -0.094,Y -539.077,Z 1232.623,A 0.000,B 0.000,C 90.000,E1 328.074} C_DIS
LIN {X -0.222,Y -534.083,Z 1232.619,A 0.000,B 0.000,C 90.000,E1 327.375} C_DIS
LIN {X -0.099,Y -527.719,Z 1232.614,A 0.000,B 0.000,C 90.000,E1 326.501} C_DIS
LIN {X 0.017,Y -517.701,Z 1232.607,A 0.000,B 0.000,C 90.000,E1 325.182} C_DIS
LIN {X -0.042,Y -515.610,Z 1232.605,A 0.000,B 0.000,C 90.000,E1 324.895} C_DIS
LIN {X -0.240,Y -512.380,Z 1232.602,A 0.000,B 0.000,C 90.000,E1 324.402} C_DIS
LIN {X -0.190,Y -510.000,Z 1232.599,A 0.000,B 0.000,C 90.000,E1 323.909} C_DIS
LIN {X 0.151,Y -507.824,Z 1232.595,A 0.000,B 0.000,C 90.000,E1 323.130} C_DIS
LIN {X 0.024,Y -506.442,Z 1232.590,A 0.000,B 0.000,C 90.000,E1 322.110} C_DIS
LIN {X -0.176,Y -506.077,Z 1232.586,A 0.000,B 0.000,C 90.000,E1 321.537} C_DIS
LIN {X -0.167,Y -506.169,Z 1232.581,A 0.000,B 0.000,C 90.000,E1 320.642} C_DIS
LIN {X -0.020,Y -507.400,Z 1232.568,A 0.000,B 0.000,C 90.000,E1 318.243} C_DIS
LIN {X 0.093,Y -508.049,Z 1232.560,A 0.000,B 0.000,C 90.000,E1 316.743} C_DIS
LIN {X -0.021,Y -508.528,Z 1232.553,A 0.000,B 0.000,C 90.000,E1 315.567} C_DIS
LIN {X -0.011,Y -509.156,Z 1232.543,A 0.000,B 0.000,C 90.000,E1 313.785} C_DIS
LIN {X 0.031,Y -509.861,Z 1232.533,A 0.000,B 0.000,C 90.000,E1 312.000} C_DIS
LIN {X -0.064,Y -510.353,Z 1232.527,A 0.000,B 0.000,C 90.000,E1 310.825} C_DIS
LIN {X -0.188,Y -510.890,Z 1232.519,A 0.000,B 0.000,C 90.000,E1 309.358} C_DIS
LIN {X -0.066,Y -511.420,Z 1232.509,A 0.000,B 0.000,C 90.000,E1 307.569} C_DIS
LIN {X -0.072,Y -511.854,Z 1232.500,A 0.000,B 0.000,C 90.000,E1 306.091} C_DIS
LIN {X -0.064,Y -512.245,Z 1232.492,A 0.000,B 0.000,C 90.000,E1 304.612} C_DIS
LIN {X -0.340,Y -512.626,Z 1232.484,A 0.000,B 0.000,C 90.000,E1 303.166} C_DIS
LIN {X 0.179,Y -512.814,Z 1232.478,A 0.000,B 0.000,C 90.000,E1 301.926} C_DIS
LIN {X -0.282,Y -512.976,Z 1232.468,A 0.000,B 0.000,C 90.000,E1 300.207} C_DIS
LIN {X -0.042,Y -513.078,Z 1232.458,A 0.000,B 0.000,C 90.000,E1 298.409} C_DIS
LIN {X 0.159,Y -513.108,Z 1232.448,A 0.000,B 0.000,C 90.000,E1 296.616} C_DIS
LIN {X -0.202,Y -513.205,Z 1232.437,A 0.000,B 0.000,C 90.000,E1 294.591} C_DIS
LIN {X 0.134,Y -513.302,Z 1232.428,A 0.000,B 0.000,C 90.000,E1 293.078} C_DIS
LIN {X 0.143,Y -513.085,Z 1232.422,A 0.000,B 0.000,C 90.000,E1 291.897} C_DIS
LIN {X -0.160,Y -512.773,Z 1232.417,A 0.000,B 0.000,C 90.000,E1 291.046} C_DIS
LIN {X -0.226,Y -512.132,Z 1232.409,A 0.000,B 0.000,C 90.000,E1 289.577} C_DIS
LIN {X 0.122,Y -511.395,Z 1232.399,A 0.000,B 0.000,C 90.000,E1 287.764} C_DIS
LIN {X -0.190,Y -510.560,Z 1232.389,A 0.000,B 0.000,C 90.000,E1 286.024} C_DIS
LIN {X -0.180,Y -510.202,Z 1232.384,A 0.000,B 0.000,C 90.000,E1 285.134} C_DIS
LIN {X -0.215,Y -508.972,Z 1232.372,A 0.000,B 0.000,C 90.000,E1 283.063} C_DIS
LIN {X 0.132,Y -507.650,Z 1232.363,A 0.000,B 0.000,C 90.000,E1 281.243} C_DIS
LIN {X 0.206,Y -506.150,Z 1232.351,A 0.000,B 0.000,C 90.000,E1 279.151} C_DIS
LIN {X 0.043,Y -505.580,Z 1232.346,A 0.000,B 0.000,C 90.000,E1 278.276} C_DIS
LIN {X -0.146,Y -504.204,Z 1232.333,A 0.000,B 0.000,C 90.000,E1 275.910} C_DIS
LIN {X 0.150,Y -503.034,Z 1232.321,A 0.000,B 0.000,C 90.000,E1 273.784} C_DIS
LIN {X -0.020,Y -501.903,Z 1232.311,A 0.000,B 0.000,C 90.000,E1 272.007} C_DIS
LIN {X 0.024,Y -500.957,Z 1232.305,A 0.000,B 0.000,C 90.000,E1 270.802} C_DIS
LIN {X -0.202,Y -499.791,Z 1232.295,A 0.000,B 0.000,C 90.000,E1 269.026} C_DIS
LIN {X -0.078,Y -498.528,Z 1232.283,A 0.000,B 0.000,C 90.000,E1 266.906} C_DIS
LIN {X -0.052,Y -497.846,Z 1232.276,A 0.000,B 0.000,C 90.000,E1 265.698} C_DIS
LIN {X -0.027,Y -497.124,Z 1232.269,A 0.000,B 0.000,C 90.000,E1 264.489} C_DIS
LIN {X -0.015,Y -496.206,Z 1232.263,A 0.000,B 0.000,C 90.000,E1 263.280} C_DIS
LIN {X 0.042,Y -495.185,Z 1232.256,A 0.000,B 0.000,C 90.000,E1 262.064} C_DIS
LIN {X -0.010,Y -493.755,Z 1232.248,A 0.000,B 0.000,C 90.000,E1 260.557} C_DIS
LIN {X 0.183,Y -491.812,Z 1232.236,A 0.000,B 0.000,C 90.000,E1 258.409} C_DIS
LIN {X -0.233,Y -490.689,Z 1232.227,A 0.000,B 0.000,C 90.000,E1 256.937} C_DIS
LIN {X -0.178,Y -489.498,Z 1232.217,A 0.000,B 0.000,C 90.000,E1 255.102} C_DIS
LIN {X -0.142,Y -488.201,Z 1232.205,A 0.000,B 0.000,C 90.000,E1 252.960} C_DIS
LIN {X 0.109,Y -487.425,Z 1232.197,A 0.000,B 0.000,C 90.000,E1 251.402} C_DIS
LIN {X 0.055,Y -486.529,Z 1232.187,A 0.000,B 0.000,C 90.000,E1 249.571} C_DIS
LIN {X 0.143,Y -485.697,Z 1232.178,A 0.000,B 0.000,C 90.000,E1 248.028} C_DIS
LIN {X 0.202,Y -484.962,Z 1232.171,A 0.000,B 0.000,C 90.000,E1 246.794} C_DIS
LIN {X 0.009,Y -483.544,Z 1232.161,A 0.000,B 0.000,C 90.000,E1 244.973} C_DIS
LIN {X -0.216,Y -482.538,Z 1232.154,A 0.000,B 0.000,C 90.000,E1 243.768} C_DIS
LIN {X 0.187,Y -481.625,Z 1232.147,A 0.000,B 0.000,C 90.000,E1 242.487} C_DIS
LIN {X -0.093,Y -479.916,Z 1232.137,A 0.000,B 0.000,C 90.000,E1 240.667} C_DIS
LIN {X -0.137,Y -478.307,Z 1232.128,A 0.000,B 0.000,C 90.000,E1 239.125} C_DIS
LIN {X 0.178,Y -476.052,Z 1232.116,A 0.000,B 0.000,C 90.000,E1 236.914} C_DIS
LIN {X -0.081,Y -474.420,Z 1232.108,A 0.000,B 0.000,C 90.000,E1 235.388} C_DIS
LIN {X 0.072,Y -472.534,Z 1232.097,A 0.000,B 0.000,C 90.000,E1 233.497} C_DIS
LIN {X -0.069,Y -471.013,Z 1232.089,A 0.000,B 0.000,C 90.000,E1 231.949} C_DIS
LIN {X -0.021,Y -469.050,Z 1232.076,A 0.000,B 0.000,C 90.000,E1 229.747} C_DIS
LIN {X 0.079,Y -467.749,Z 1232.068,A 0.000,B 0.000,C 90.000,E1 228.162} C_DIS
LIN {X -0.131,Y -466.250,Z 1232.057,A 0.000,B 0.000,C 90.000,E1 226.296} C_DIS
LIN {X -0.027,Y -463.890,Z 1232.027,A 0.000,B 0.000,C 90.000,E1 220.906} C_DIS
LIN {X 0.001,Y -465.266,Z 1231.997,A 0.000,B 0.000,C 90.000,E1 215.518} C_DIS
LIN {X 0.006,Y -466.949,Z 1231.982,A 0.000,B 0.000,C 90.000,E1 212.673} C_DIS
LIN {X -0.114,Y -468.755,Z 1231.971,A 0.000,B 0.000,C 90.000,E1 210.797} C_DIS
LIN {X -0.157,Y -471.784,Z 1231.955,A 0.000,B 0.000,C 90.000,E1 207.975} C_DIS
LIN {X -0.077,Y -474.896,Z 1231.941,A 0.000,B 0.000,C 90.000,E1 205.463} C_DIS
LIN {X 0.067,Y -480.490,Z 1231.921,A 0.000,B 0.000,C 90.000,E1 201.716} C_DIS
LIN {X 0.246,Y -488.129,Z 1231.899,A 0.000,B 0.000,C 90.000,E1 197.692} C_DIS
LIN {X 0.208,Y -494.468,Z 1231.883,A 0.000,B 0.000,C 90.000,E1 194.954} C_DIS
LIN {X -0.106,Y -499.031,Z 1231.873,A 0.000,B 0.000,C 90.000,E1 193.175} C_DIS
LIN {X 0.009,Y -502.924,Z 1231.865,A 0.000,B 0.000,C 90.000,E1 191.658} C_DIS
LIN {X 0.017,Y -510.293,Z 1231.850,A 0.000,B 0.000,C 90.000,E1 188.973} C_DIS
LIN {X 0.194,Y -514.474,Z 1231.842,A 0.000,B 0.000,C 90.000,E1 187.473} C_DIS
LIN {X -0.055,Y -518.520,Z 1231.833,A 0.000,B 0.000,C 90.000,E1 186.030} C_DIS
LIN {X -0.240,Y -522.595,Z 1231.825,A 0.000,B 0.000,C 90.000,E1 184.588} C_DIS
LIN {X 0.081,Y -527.453,Z 1231.816,A 0.000,B 0.000,C 90.000,E1 182.808} C_DIS
LIN {X -0.027,Y -531.498,Z 1231.808,A 0.000,B 0.000,C 90.000,E1 181.375} C_DIS
LIN {X -0.070,Y -537.003,Z 1231.797,A 0.000,B 0.000,C 90.000,E1 179.370} C_DIS
LIN {X -0.036,Y -540.040,Z 1231.790,A 0.000,B 0.000,C 90.000,E1 178.224} C_DIS
LIN {X 0.111,Y -543.728,Z 1231.782,A 0.000,B 0.000,C 90.000,E1 176.788} C_DIS
LIN {X -0.170,Y -547.899,Z 1231.773,A 0.000,B 0.000,C 90.000,E1 175.122} C_DIS
LIN {X 0.130,Y -551.245,Z 1231.765,A 0.000,B 0.000,C 90.000,E1 173.685} C_DIS
LIN {X 0.160,Y -555.728,Z 1231.754,A 0.000,B 0.000,C 90.000,E1 171.724} C_DIS
LIN {X 0.183,Y -558.838,Z 1231.746,A 0.000,B 0.000,C 90.000,E1 170.330} C_DIS
LIN {X 0.213,Y -561.323,Z 1231.740,A 0.000,B 0.000,C 90.000,E1 169.218} C_DIS
LIN {X -0.060,Y -564.905,Z 1231.731,A 0.000,B 0.000,C 90.000,E1 167.589} C_DIS
LIN {X -0.193,Y -567.999,Z 1231.723,A 0.000,B 0.000,C 90.000,E1 166.228} C_DIS
LIN {X -0.285,Y -574.465,Z 1231.708,A 0.000,B 0.000,C 90.000,E1 163.504} C_DIS
LIN {X -0.038,Y -581.367,Z 1231.695,A 0.000,B 0.000,C 90.000,E1 161.040} C_DIS
LIN {X -0.143,Y -588.854,Z 1231.683,A 0.000,B 0.000,C 90.000,E1 158.901} C_DIS
LIN {X 0.187,Y -597.580,Z 1231.671,A 0.000,B 0.000,C 90.000,E1 156.741} C_DIS
LIN {X 0.088,Y -603.058,Z 1231.664,A 0.000,B 0.000,C 90.000,E1 155.433} C_DIS
